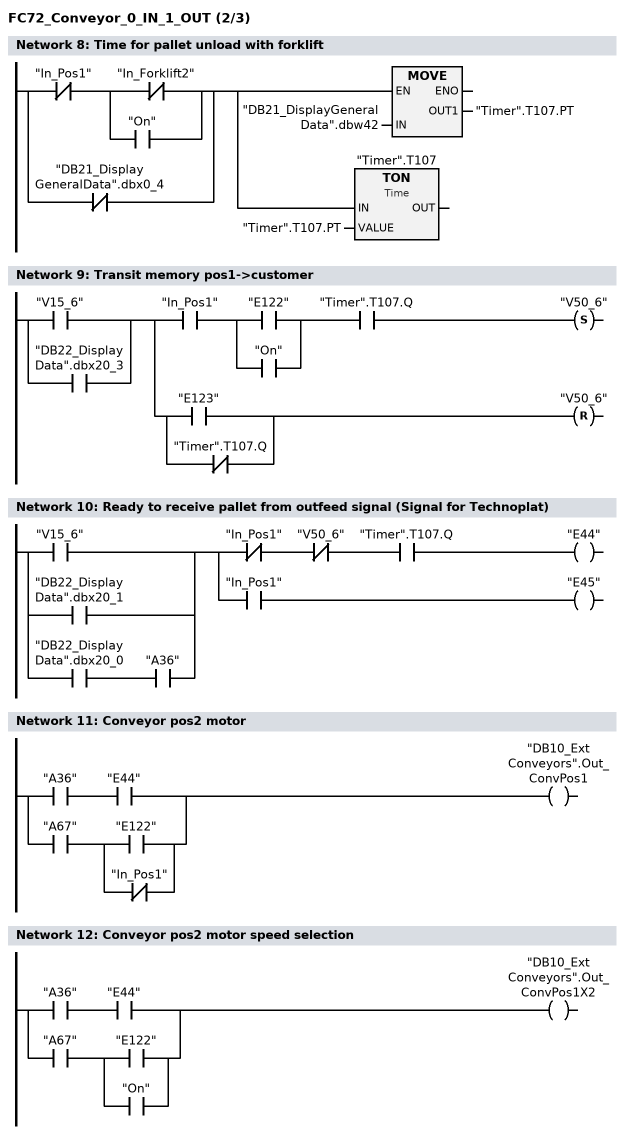
   #_w1 := (NOT "In_Pos1" AND (NOT "In_Forklift2" OR "On")) OR NOT "DB21_DisplayGeneralData".dbx0_4;
   IF #_w1 THEN "Timer".T107.PT := "DB21_DisplayGeneralData".dbw42; END_IF;
   "Timer".T107.TON(IN := #_w1, PT := "Timer".T107.PT);   // TON coil
END_REGION

REGION Network 9: Transit memory pos1->customer
   RUNG wire#powerrail
      Contact( "V15_6" )
      wire#w1
      Contact( "In_Pos1" )
      wire#w2
      Contact( "E122" )
      wire#w3
      Contact( "Timer".T107.Q )
      S_Coil( "V50_6" )
   END_RUNG
   RUNG wire#powerrail
      Contact( "DB22_DisplayData".dbx20_3 )
   END_RUNG wire#w1
   RUNG wire#w2
      Contact( "On" )
   END_RUNG wire#w3
   RUNG wire#w1
      Contact( "E123" )
      wire#w4
      R_Coil( "V50_6" )
   END_RUNG
   RUNG wire#w1
      I_Contact( "Timer".T107.Q )
   END_RUNG wire#w4
   // the same network as SCL:
   #_w1 := "V15_6" OR "DB22_DisplayData".dbx20_3;
   IF #_w1 AND "In_Pos1" AND ("E122" OR "On") AND "Timer".T107.Q THEN "V50_6" := TRUE; END_IF;
   IF #_w1 AND ("E123" OR NOT "Timer".T107.Q) THEN "V50_6" := FALSE; END_IF;
END_REGION

REGION Network 10: Ready to receive pallet from outfeed signal (Signal for Technoplat)
   RUNG wire#powerrail
      Contact( "V15_6" )
      wire#w1
      I_Contact( "In_Pos1" )
      I_Contact( "V50_6" )
      Contact( "Timer".T107.Q )
      Coil( "E44" )
   END_RUNG
   RUNG wire#powerrail
      Contact( "DB22_DisplayData".dbx20_1 )
   END_RUNG wire#w1
   RUNG wire#powerrail
      Contact( "DB22_DisplayData".dbx20_0 )
      Contact( "A36" )
   END_RUNG wire#w1
   RUNG wire#w1
      Contact( "In_Pos1" )
      Coil( "E45" )
   END_RUNG
   // the same network as SCL:
   #_w1 := "V15_6" OR "DB22_DisplayData".dbx20_1 OR ("DB22_DisplayData".dbx20_0 AND "A36");
   "E44" := #_w1 AND NOT "In_Pos1" AND NOT "V50_6" AND "Timer".T107.Q;
   "E45" := #_w1 AND "In_Pos1";
END_REGION

REGION Network 11: Conveyor pos2 motor
   RUNG wire#powerrail
      Contact( "A36" )
      Contact( "E44" )
      wire#w1
      Coil( "DB10_ExtConveyors".Out_ConvPos1 )
   END_RUNG
   RUNG wire#powerrail
      Contact( "A67" )
      wire#w2
      Contact( "E122" )
   END_RUNG wire#w1
   RUNG wire#w2
      I_Contact( "In_Pos1" )
   END_RUNG wire#w1
   // the same network as SCL:
   "DB10_ExtConveyors".Out_ConvPos1 := ("A36" AND "E44") OR ("A67" AND ("E122" OR NOT "In_Pos1"));
END_REGION

REGION Network 12: Conveyor pos2 motor speed selection
   RUNG wire#powerrail
      Contact( "A36" )
      Contact( "E44" )
      wire#w1
      Coil( "DB10_ExtConveyors".Out_ConvPos1X2 )
   END_RUNG
   RUNG wire#powerrail
      Contact( "A67" )
      wire#w2
      Contact( "E122" )
   END_RUNG wire#w1
   RUNG wire#w2
      Contact( "On" )
   END_RUNG wire#w1
   // the same network as SCL:
   "DB10_ExtConveyors".Out_ConvPos1X2 := ("A36" AND "E44") OR ("A67" AND ("E122" OR "On"));
END_REGION

REGION Network 13: Pallet ready in outfeed signal
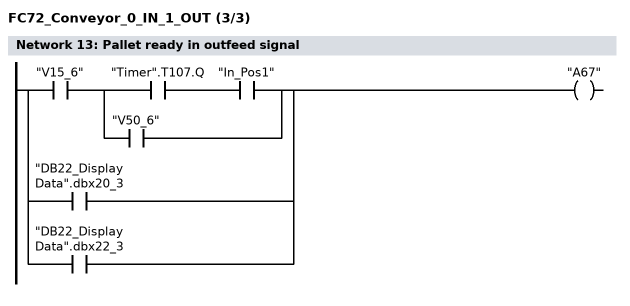
   RUNG wire#powerrail
      Contact( "V15_6" )
      wire#w1
      Contact( "Timer".T107.Q )
      Contact( "In_Pos1" )
      wire#w2
      Coil( "A67" )
   END_RUNG
   RUNG wire#w1
      Contact( "V50_6" )
   END_RUNG wire#w2
   RUNG wire#powerrail
      Contact( "DB22_DisplayData".dbx20_3 )
   END_RUNG wire#w2
   RUNG wire#powerrail
      Contact( "DB22_DisplayData".dbx22_3 )
   END_RUNG wire#w2
   // the same network as SCL:
   "A67" := ("V15_6" AND (("Timer".T107.Q AND "In_Pos1") OR "V50_6")) OR "DB22_DisplayData".dbx20_3 OR "DB22_DisplayData".dbx22_3;
END_REGION
END_FUNCTION

FUNCTION "FC37_MultiprogramSignal" : Void   // FC37, LAD
TITLE = Multiprogram with program selection by external signal
{ S7_Optimized_Access := 'FALSE' }
AUTHOR : Robopac
VERSION : 0.0
// stored: AutoNumber false, IsIECCheckEnabled false, SetENOAutomatically false, UDAEnableTagReadback false
   VAR_TEMP   // added for the SCL form of the ladder/FBD networks
      _w1 : Bool;
   END_VAR
BEGIN

REGION Network 1
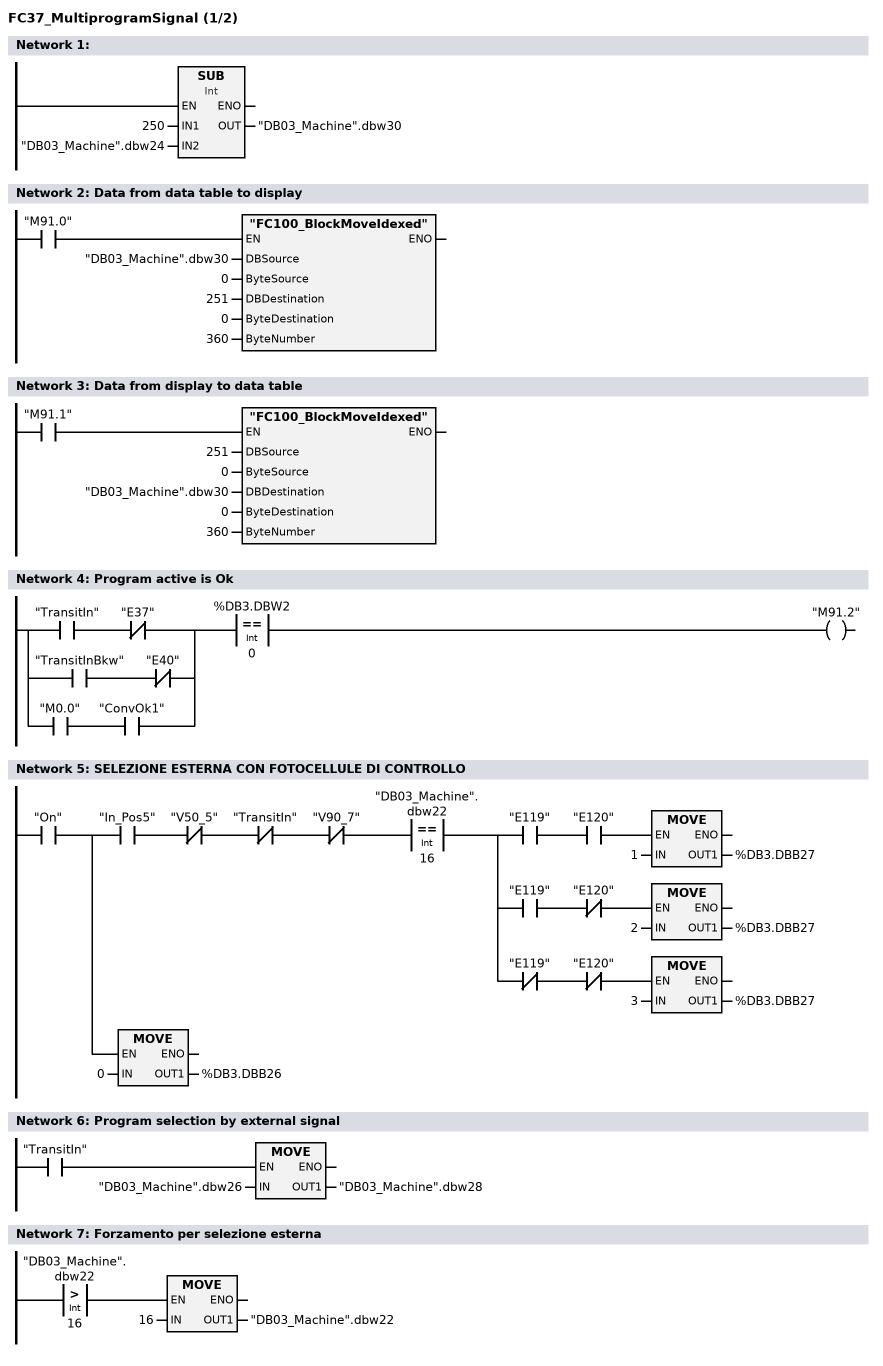
   RUNG wire#powerrail
      { S7_Templates := "SrcType := Int"; S7_GenerateENO := "TRUE" } Sub(in1 := 250, in2 := "DB03_Machine".dbw24, out => "DB03_Machine".dbw30)
   END_RUNG
   // the same network as SCL:
   "DB03_Machine".dbw30 := 250 - "DB03_Machine".dbw24;
END_REGION

REGION Network 2: Data from data table to display
   RUNG wire#powerrail
      Contact( "M91.0" )
      "FC100_BlockMoveIdexed"(DBSource := "DB03_Machine".dbw30, ByteSource := 0, DBDestination := 251, ByteDestination := 0, ByteNumber := 360)
   END_RUNG
   // the same network as SCL:
   IF "M91.0" THEN
       "FC100_BlockMoveIdexed"(DBSource := "DB03_Machine".dbw30,
                               ByteSource := 0,
                               DBDestination := 251,
                               ByteDestination := 0,
                               ByteNumber := 360);
   END_IF;
END_REGION

REGION Network 3: Data from display to data table
   RUNG wire#powerrail
      Contact( "M91.1" )
      "FC100_BlockMoveIdexed"(DBSource := 251, ByteSource := 0, DBDestination := "DB03_Machine".dbw30, ByteDestination := 0, ByteNumber := 360)
   END_RUNG
   // the same network as SCL:
   IF "M91.1" THEN
       "FC100_BlockMoveIdexed"(DBSource := 251,
                               ByteSource := 0,
                               DBDestination := "DB03_Machine".dbw30,
                               ByteDestination := 0,
                               ByteNumber := 360);
   END_IF;
END_REGION

REGION Network 4: Program active is Ok
   RUNG wire#powerrail
      Contact( "TransitIn" )
      I_Contact( "E37" )
      wire#w1
      { S7_Templates := "SrcType := Int" } EQ_Contact(in1 := %DB3.DBW2, in2 := 0)
      Coil( "M91.2" )
   END_RUNG
   RUNG wire#powerrail
      Contact( "TransitInBkw" )
      I_Contact( "E40" )
   END_RUNG wire#w1
   RUNG wire#powerrail
      Contact( "M0.0" )
      Contact( "ConvOk1" )
   END_RUNG wire#w1
   // the same network as SCL:
   "M91.2" := (("TransitIn" AND NOT "E37") OR ("TransitInBkw" AND NOT "E40") OR ("M0.0" AND "ConvOk1")) AND (%DB3.DBW2 = 0);
END_REGION

REGION Network 5: SELEZIONE ESTERNA CON FOTOCELLULE DI CONTROLLO
   RUNG wire#powerrail
      Contact( "On" )
      wire#w1
      Contact( "In_Pos5" )
      I_Contact( "V50_5" )
      I_Contact( "TransitIn" )
      I_Contact( "V90_7" )
      { S7_Templates := "SrcType := Int" } EQ_Contact(in1 := "DB03_Machine".dbw22, in2 := 16)
      wire#w2
      Contact( "E119" )
      Contact( "E120" )
      Move(in := 1, out1 => %DB3.DBB27)
   END_RUNG
   RUNG wire#w2
      Contact( "E119" )
      I_Contact( "E120" )
      Move(in := 2, out1 => %DB3.DBB27)
   END_RUNG
   RUNG wire#w2
      I_Contact( "E119" )
      I_Contact( "E120" )
      Move(in := 3, out1 => %DB3.DBB27)
   END_RUNG
   RUNG wire#w1
      { S7_GenerateENO := "TRUE" } Move(in := 0, out1 => %DB3.DBB26)
   END_RUNG
   // the same network as SCL:
   #_w1 := "On" AND "In_Pos5" AND NOT "V50_5" AND NOT "TransitIn" AND NOT "V90_7" AND ("DB03_Machine".dbw22 = 16);
   IF #_w1 AND "E119" AND "E120" THEN %DB3.DBB27 := 1; END_IF;
   IF #_w1 AND "E119" AND NOT "E120" THEN %DB3.DBB27 := 2; END_IF;
   IF #_w1 AND NOT "E119" AND NOT "E120" THEN %DB3.DBB27 := 3; END_IF;
   IF "On" THEN %DB3.DBB26 := 0; END_IF;
END_REGION

REGION Network 6: Program selection by external signal
   RUNG wire#powerrail
      Contact( "TransitIn" )
      { S7_GenerateENO := "TRUE" } Move(in := "DB03_Machine".dbw26, out1 => "DB03_Machine".dbw28)
   END_RUNG
   // the same network as SCL:
   IF "TransitIn" THEN "DB03_Machine".dbw28 := "DB03_Machine".dbw26; END_IF;
END_REGION

REGION Network 7: Forzamento per selezione esterna
   RUNG wire#powerrail
      { S7_Templates := "SrcType := Int" } GT_Contact(in1 := "DB03_Machine".dbw22, in2 := 16)
      { S7_GenerateENO := "TRUE" } Move(in := 16, out1 => "DB03_Machine".dbw22)
   END_RUNG
   // the same network as SCL:
   IF "DB03_Machine".dbw22 > 16 THEN "DB03_Machine".dbw22 := 16; END_IF;
END_REGION

REGION Network 8: Program selection by display
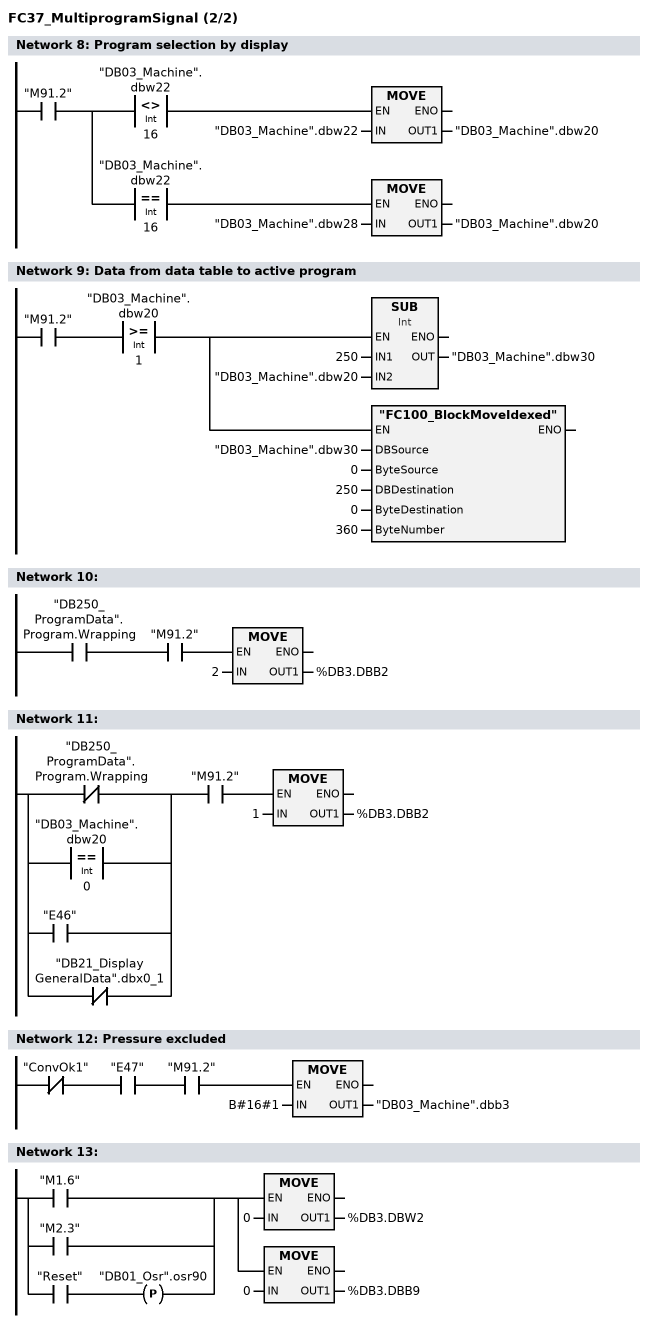
   RUNG wire#powerrail
      Contact( "M91.2" )
      wire#w1
      { S7_Templates := "SrcType := Int" } NE_Contact(in1 := "DB03_Machine".dbw22, in2 := 16)
      { S7_GenerateENO := "TRUE" } Move(in := "DB03_Machine".dbw22, out1 => "DB03_Machine".dbw20)
   END_RUNG
   RUNG wire#w1
      { S7_Templates := "SrcType := Int" } EQ_Contact(in1 := "DB03_Machine".dbw22, in2 := 16)
      { S7_GenerateENO := "TRUE" } Move(in := "DB03_Machine".dbw28, out1 => "DB03_Machine".dbw20)
   END_RUNG
   // the same network as SCL:
   IF "M91.2" AND ("DB03_Machine".dbw22 <> 16) THEN "DB03_Machine".dbw20 := "DB03_Machine".dbw22; END_IF;
   IF "M91.2" AND ("DB03_Machine".dbw22 = 16) THEN "DB03_Machine".dbw20 := "DB03_Machine".dbw28; END_IF;
END_REGION

REGION Network 9: Data from data table to active program
   RUNG wire#powerrail
      Contact( "M91.2" )
      { S7_Templates := "SrcType := Int" } GE_Contact(in1 := "DB03_Machine".dbw20, in2 := 1)
      wire#w1
      { S7_Templates := "SrcType := Int"; S7_GenerateENO := "TRUE" } Sub(in1 := 250, in2 := "DB03_Machine".dbw20, out => "DB03_Machine".dbw30)
   END_RUNG
   RUNG wire#w1
      "FC100_BlockMoveIdexed"(DBSource := "DB03_Machine".dbw30, ByteSource := 0, DBDestination := 250, ByteDestination := 0, ByteNumber := 360)
   END_RUNG
   // the same network as SCL:
   IF "M91.2" AND ("DB03_Machine".dbw20 >= 1) THEN
       "DB03_Machine".dbw30 := 250 - "DB03_Machine".dbw20;
       "FC100_BlockMoveIdexed"(DBSource := "DB03_Machine".dbw30,
                               ByteSource := 0,
                               DBDestination := 250,
                               ByteDestination := 0,
                               ByteNumber := 360);
   END_IF;
END_REGION

REGION Network 10
   RUNG wire#powerrail
      Contact( "DB250_ProgramData".Program.Wrapping )
      Contact( "M91.2" )
      { S7_GenerateENO := "TRUE" } Move(in := 2, out1 => %DB3.DBB2)
   END_RUNG
   // the same network as SCL:
   IF "DB250_ProgramData".Program.Wrapping AND "M91.2" THEN %DB3.DBB2 := 2; END_IF;
END_REGION

REGION Network 11
   RUNG wire#powerrail
      I_Contact( "DB250_ProgramData".Program.Wrapping )
      wire#w1
      Contact( "M91.2" )
      { S7_GenerateENO := "TRUE" } Move(in := 1, out1 => %DB3.DBB2)
   END_RUNG
   RUNG wire#powerrail
      { S7_Templates := "SrcType := Int" } EQ_Contact(in1 := "DB03_Machine".dbw20, in2 := 0)
   END_RUNG wire#w1
   RUNG wire#powerrail
      Contact( "E46" )
   END_RUNG wire#w1
   RUNG wire#powerrail
      I_Contact( "DB21_DisplayGeneralData".dbx0_1 )
   END_RUNG wire#w1
   // the same network as SCL:
   IF (NOT "DB250_ProgramData".Program.Wrapping OR ("DB03_Machine".dbw20 = 0) OR "E46" OR NOT "DB21_DisplayGeneralData".dbx0_1) AND "M91.2" THEN
       %DB3.DBB2 := 1;
   END_IF;
END_REGION

REGION Network 12: Pressure excluded
   RUNG wire#powerrail
      I_Contact( "ConvOk1" )
      Contact( "E47" )
      Contact( "M91.2" )
      { S7_GenerateENO := "TRUE" } Move(in := B#16#1, out1 => "DB03_Machine".dbb3)
   END_RUNG
   // the same network as SCL:
   IF NOT "ConvOk1" AND "E47" AND "M91.2" THEN "DB03_Machine".dbb3 := B#16#1; END_IF;
END_REGION

REGION Network 13
   RUNG wire#powerrail
      Contact( "M1.6" )
      wire#w1
      { S7_GenerateENO := "TRUE" } Move(in := 0, out1 => %DB3.DBW2)
   END_RUNG
   RUNG wire#powerrail
      Contact( "M2.3" )
   END_RUNG wire#w1
   RUNG wire#powerrail
      Contact( "Reset" )
      P_Trig( "DB01_Osr".osr90 )
   END_RUNG wire#w1
   RUNG wire#w1
      { S7_GenerateENO := "TRUE" } Move(in := 0, out1 => %DB3.DBB9)
   END_RUNG
   // the same network as SCL:
   #_w1 := "Reset" AND NOT "DB01_Osr".osr90;   // rising edge
   "DB01_Osr".osr90 := "Reset";
   IF "M1.6" OR "M2.3" OR #_w1 THEN
       %DB3.DBW2 := 0;
       %DB3.DBB9 := 0;
   END_IF;
END_REGION
END_FUNCTION

FUNCTION "FC39_DisplaySiemensTP" : Void   // FC39, LAD
TITLE = Display Siemens TP177 management
{ S7_Optimized_Access := 'FALSE' }
AUTHOR : Robopac
VERSION : 0.0
// stored: AutoNumber false, IsIECCheckEnabled false, SetENOAutomatically false, UDAEnableTagReadback false
   VAR_TEMP
      TempInt : Int;
   END_VAR
   VAR_TEMP   // added for the SCL form of the ladder/FBD networks
      _w1 : Bool;
      _w2 : Bool;
      _w3 : Bool;
      _w4 : Bool;
      _w5 : Bool;
      _w6 : Bool;
   END_VAR
BEGIN

REGION Network 1: Manual(Toggle bit): Pressure plate upward/downward (Helix)
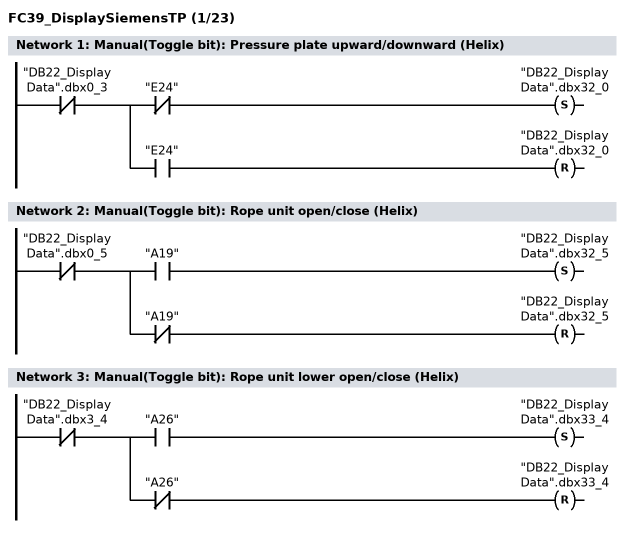
   RUNG wire#powerrail
      I_Contact( "DB22_DisplayData".dbx0_3 )
      wire#w1
      I_Contact( "E24" )
      S_Coil( "DB22_DisplayData".dbx32_0 )
   END_RUNG
   RUNG wire#w1
      Contact( "E24" )
      R_Coil( "DB22_DisplayData".dbx32_0 )
   END_RUNG
   // the same network as SCL:
   #_w1 := NOT "DB22_DisplayData".dbx0_3;
   IF #_w1 AND NOT "E24" THEN "DB22_DisplayData".dbx32_0 := TRUE; END_IF;
   IF #_w1 AND "E24" THEN "DB22_DisplayData".dbx32_0 := FALSE; END_IF;
END_REGION

REGION Network 2: Manual(Toggle bit): Rope unit open/close (Helix)
   RUNG wire#powerrail
      I_Contact( "DB22_DisplayData".dbx0_5 )
      wire#w1
      Contact( "A19" )
      S_Coil( "DB22_DisplayData".dbx32_5 )
   END_RUNG
   RUNG wire#w1
      I_Contact( "A19" )
      R_Coil( "DB22_DisplayData".dbx32_5 )
   END_RUNG
   // the same network as SCL:
   #_w1 := NOT "DB22_DisplayData".dbx0_5;
   IF #_w1 AND "A19" THEN "DB22_DisplayData".dbx32_5 := TRUE; END_IF;
   IF #_w1 AND NOT "A19" THEN "DB22_DisplayData".dbx32_5 := FALSE; END_IF;
END_REGION

REGION Network 3: Manual(Toggle bit): Rope unit lower open/close (Helix)
   RUNG wire#powerrail
      I_Contact( "DB22_DisplayData".dbx3_4 )
      wire#w1
      Contact( "A26" )
      S_Coil( "DB22_DisplayData".dbx33_4 )
   END_RUNG
   RUNG wire#w1
      I_Contact( "A26" )
      R_Coil( "DB22_DisplayData".dbx33_4 )
   END_RUNG
   // the same network as SCL:
   #_w1 := NOT "DB22_DisplayData".dbx3_4;
   IF #_w1 AND "A26" THEN "DB22_DisplayData".dbx33_4 := TRUE; END_IF;
   IF #_w1 AND NOT "A26" THEN "DB22_DisplayData".dbx33_4 := FALSE; END_IF;
END_REGION

REGION Network 4: Manual operation for Helix
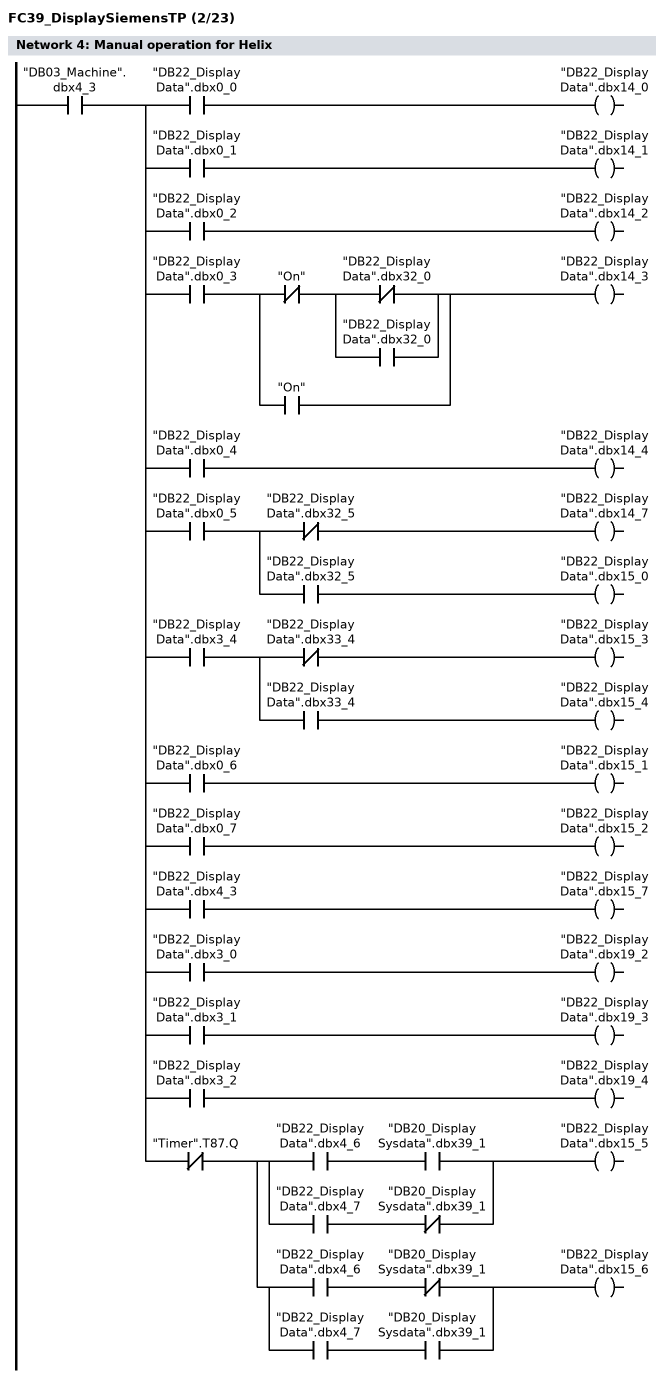
   RUNG wire#powerrail
      Contact( "DB03_Machine".dbx4_3 )
      wire#w1
      Contact( "DB22_DisplayData".dbx0_0 )
      Coil( "DB22_DisplayData".dbx14_0 )
   END_RUNG
   RUNG wire#w1
      Contact( "DB22_DisplayData".dbx0_1 )
      Coil( "DB22_DisplayData".dbx14_1 )
   END_RUNG
   RUNG wire#w1
      Contact( "DB22_DisplayData".dbx0_2 )
      Coil( "DB22_DisplayData".dbx14_2 )
   END_RUNG
   RUNG wire#w1
      Contact( "DB22_DisplayData".dbx0_3 )
      wire#w2
      I_Contact( "On" )
      wire#w3
      I_Contact( "DB22_DisplayData".dbx32_0 )
      wire#w4
      Coil( "DB22_DisplayData".dbx14_3 )
   END_RUNG
   RUNG wire#w3
      Contact( "DB22_DisplayData".dbx32_0 )
   END_RUNG wire#w4
   RUNG wire#w2
      Contact( "On" )
   END_RUNG wire#w4
   RUNG wire#w1
      Contact( "DB22_DisplayData".dbx0_4 )
      Coil( "DB22_DisplayData".dbx14_4 )
   END_RUNG
   RUNG wire#w1
      Contact( "DB22_DisplayData".dbx0_5 )
      wire#w5
      I_Contact( "DB22_DisplayData".dbx32_5 )
      Coil( "DB22_DisplayData".dbx14_7 )
   END_RUNG
   RUNG wire#w5
      Contact( "DB22_DisplayData".dbx32_5 )
      Coil( "DB22_DisplayData".dbx15_0 )
   END_RUNG
   RUNG wire#w1
      Contact( "DB22_DisplayData".dbx3_4 )
      wire#w6
      I_Contact( "DB22_DisplayData".dbx33_4 )
      Coil( "DB22_DisplayData".dbx15_3 )
   END_RUNG
   RUNG wire#w6
      Contact( "DB22_DisplayData".dbx33_4 )
      Coil( "DB22_DisplayData".dbx15_4 )
   END_RUNG
   RUNG wire#w1
      Contact( "DB22_DisplayData".dbx0_6 )
      Coil( "DB22_DisplayData".dbx15_1 )
   END_RUNG
   RUNG wire#w1
      Contact( "DB22_DisplayData".dbx0_7 )
      Coil( "DB22_DisplayData".dbx15_2 )
   END_RUNG
   RUNG wire#w1
      Contact( "DB22_DisplayData".dbx4_3 )
      Coil( "DB22_DisplayData".dbx15_7 )
   END_RUNG
   RUNG wire#w1
      Contact( "DB22_DisplayData".dbx3_0 )
      Coil( "DB22_DisplayData".dbx19_2 )
   END_RUNG
   RUNG wire#w1
      Contact( "DB22_DisplayData".dbx3_1 )
      Coil( "DB22_DisplayData".dbx19_3 )
   END_RUNG
   RUNG wire#w1
      Contact( "DB22_DisplayData".dbx3_2 )
      Coil( "DB22_DisplayData".dbx19_4 )
   END_RUNG
   RUNG wire#w1
      I_Contact( "Timer".T87.Q )
      wire#w7
      Contact( "DB22_DisplayData".dbx4_6 )
      Contact( "DB20_DisplaySysdata".dbx39_1 )
      wire#w8
      Coil( "DB22_DisplayData".dbx15_5 )
   END_RUNG
   RUNG wire#w7
      Contact( "DB22_DisplayData".dbx4_7 )
      I_Contact( "DB20_DisplaySysdata".dbx39_1 )
   END_RUNG wire#w8
   RUNG wire#w7
      Contact( "DB22_DisplayData".dbx4_6 )
      I_Contact( "DB20_DisplaySysdata".dbx39_1 )
      wire#w9
      Coil( "DB22_DisplayData".dbx15_6 )
   END_RUNG
   RUNG wire#w7
      Contact( "DB22_DisplayData".dbx4_7 )
      Contact( "DB20_DisplaySysdata".dbx39_1 )
   END_RUNG wire#w9
   // the same network as SCL:
   "DB22_DisplayData".dbx14_0 := "DB03_Machine".dbx4_3 AND "DB22_DisplayData".dbx0_0;
   "DB22_DisplayData".dbx14_1 := "DB03_Machine".dbx4_3 AND "DB22_DisplayData".dbx0_1;
   "DB22_DisplayData".dbx14_2 := "DB03_Machine".dbx4_3 AND "DB22_DisplayData".dbx0_2;
   "DB22_DisplayData".dbx14_3 := "DB03_Machine".dbx4_3 AND "DB22_DisplayData".dbx0_3 AND ((NOT "On" AND (NOT "DB22_DisplayData".dbx32_0 OR "DB22_DisplayData".dbx32_0)) OR "On");
   "DB22_DisplayData".dbx14_4 := "DB03_Machine".dbx4_3 AND "DB22_DisplayData".dbx0_4;
   #_w1 := "DB03_Machine".dbx4_3 AND "DB22_DisplayData".dbx0_5;
   "DB22_DisplayData".dbx14_7 := #_w1 AND NOT "DB22_DisplayData".dbx32_5;
   "DB22_DisplayData".dbx15_0 := #_w1 AND "DB22_DisplayData".dbx32_5;
   #_w2 := "DB03_Machine".dbx4_3 AND "DB22_DisplayData".dbx3_4;
   "DB22_DisplayData".dbx15_3 := #_w2 AND NOT "DB22_DisplayData".dbx33_4;
   "DB22_DisplayData".dbx15_4 := #_w2 AND "DB22_DisplayData".dbx33_4;
   "DB22_DisplayData".dbx15_1 := "DB03_Machine".dbx4_3 AND "DB22_DisplayData".dbx0_6;
   "DB22_DisplayData".dbx15_2 := "DB03_Machine".dbx4_3 AND "DB22_DisplayData".dbx0_7;
   "DB22_DisplayData".dbx15_7 := "DB03_Machine".dbx4_3 AND "DB22_DisplayData".dbx4_3;
   "DB22_DisplayData".dbx19_2 := "DB03_Machine".dbx4_3 AND "DB22_DisplayData".dbx3_0;
   "DB22_DisplayData".dbx19_3 := "DB03_Machine".dbx4_3 AND "DB22_DisplayData".dbx3_1;
   "DB22_DisplayData".dbx19_4 := "DB03_Machine".dbx4_3 AND "DB22_DisplayData".dbx3_2;
   #_w3 := "DB03_Machine".dbx4_3 AND NOT "Timer".T87.Q;
   "DB22_DisplayData".dbx15_5 := #_w3 AND (("DB22_DisplayData".dbx4_6 AND "DB20_DisplaySysdata".dbx39_1) OR ("DB22_DisplayData".dbx4_7 AND NOT "DB20_DisplaySysdata".dbx39_1));
   "DB22_DisplayData".dbx15_6 := #_w3 AND (("DB22_DisplayData".dbx4_6 AND NOT "DB20_DisplaySysdata".dbx39_1) OR ("DB22_DisplayData".dbx4_7 AND "DB20_DisplaySysdata".dbx39_1));
END_REGION

REGION Network 5: Manual(Toggle bit): Clamp upward/downward (Clamp)
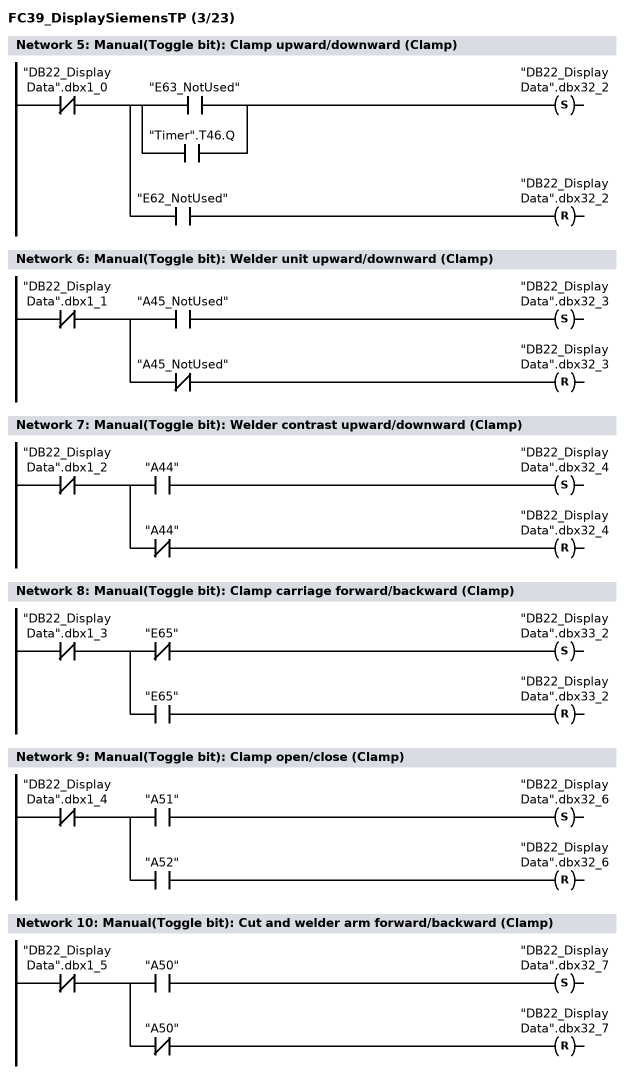
   RUNG wire#powerrail
      I_Contact( "DB22_DisplayData".dbx1_0 )
      wire#w1
      Contact( "E63_NotUsed" )
      wire#w2
      S_Coil( "DB22_DisplayData".dbx32_2 )
   END_RUNG
   RUNG wire#w1
      Contact( "Timer".T46.Q )
   END_RUNG wire#w2
   RUNG wire#w1
      Contact( "E62_NotUsed" )
      R_Coil( "DB22_DisplayData".dbx32_2 )
   END_RUNG
   // the same network as SCL:
   #_w1 := NOT "DB22_DisplayData".dbx1_0;
   IF #_w1 AND ("E63_NotUsed" OR "Timer".T46.Q) THEN "DB22_DisplayData".dbx32_2 := TRUE; END_IF;
   IF #_w1 AND "E62_NotUsed" THEN "DB22_DisplayData".dbx32_2 := FALSE; END_IF;
END_REGION

REGION Network 6: Manual(Toggle bit): Welder unit upward/downward (Clamp)
   RUNG wire#powerrail
      I_Contact( "DB22_DisplayData".dbx1_1 )
      wire#w1
      Contact( "A45_NotUsed" )
      S_Coil( "DB22_DisplayData".dbx32_3 )
   END_RUNG
   RUNG wire#w1
      I_Contact( "A45_NotUsed" )
      R_Coil( "DB22_DisplayData".dbx32_3 )
   END_RUNG
   // the same network as SCL:
   #_w1 := NOT "DB22_DisplayData".dbx1_1;
   IF #_w1 AND "A45_NotUsed" THEN "DB22_DisplayData".dbx32_3 := TRUE; END_IF;
   IF #_w1 AND NOT "A45_NotUsed" THEN "DB22_DisplayData".dbx32_3 := FALSE; END_IF;
END_REGION

REGION Network 7: Manual(Toggle bit): Welder contrast upward/downward (Clamp)
   RUNG wire#powerrail
      I_Contact( "DB22_DisplayData".dbx1_2 )
      wire#w1
      Contact( "A44" )
      S_Coil( "DB22_DisplayData".dbx32_4 )
   END_RUNG
   RUNG wire#w1
      I_Contact( "A44" )
      R_Coil( "DB22_DisplayData".dbx32_4 )
   END_RUNG
   // the same network as SCL:
   #_w1 := NOT "DB22_DisplayData".dbx1_2;
   IF #_w1 AND "A44" THEN "DB22_DisplayData".dbx32_4 := TRUE; END_IF;
   IF #_w1 AND NOT "A44" THEN "DB22_DisplayData".dbx32_4 := FALSE; END_IF;
END_REGION

REGION Network 8: Manual(Toggle bit): Clamp carriage forward/backward (Clamp)
   RUNG wire#powerrail
      I_Contact( "DB22_DisplayData".dbx1_3 )
      wire#w1
      I_Contact( "E65" )
      S_Coil( "DB22_DisplayData".dbx33_2 )
   END_RUNG
   RUNG wire#w1
      Contact( "E65" )
      R_Coil( "DB22_DisplayData".dbx33_2 )
   END_RUNG
   // the same network as SCL:
   #_w1 := NOT "DB22_DisplayData".dbx1_3;
   IF #_w1 AND NOT "E65" THEN "DB22_DisplayData".dbx33_2 := TRUE; END_IF;
   IF #_w1 AND "E65" THEN "DB22_DisplayData".dbx33_2 := FALSE; END_IF;
END_REGION

REGION Network 9: Manual(Toggle bit): Clamp open/close (Clamp)
   RUNG wire#powerrail
      I_Contact( "DB22_DisplayData".dbx1_4 )
      wire#w1
      Contact( "A51" )
      S_Coil( "DB22_DisplayData".dbx32_6 )
   END_RUNG
   RUNG wire#w1
      Contact( "A52" )
      R_Coil( "DB22_DisplayData".dbx32_6 )
   END_RUNG
   // the same network as SCL:
   #_w1 := NOT "DB22_DisplayData".dbx1_4;
   IF #_w1 AND "A51" THEN "DB22_DisplayData".dbx32_6 := TRUE; END_IF;
   IF #_w1 AND "A52" THEN "DB22_DisplayData".dbx32_6 := FALSE; END_IF;
END_REGION

REGION Network 10: Manual(Toggle bit): Cut and welder arm forward/backward (Clamp)
   RUNG wire#powerrail
      I_Contact( "DB22_DisplayData".dbx1_5 )
      wire#w1
      Contact( "A50" )
      S_Coil( "DB22_DisplayData".dbx32_7 )
   END_RUNG
   RUNG wire#w1
      I_Contact( "A50" )
      R_Coil( "DB22_DisplayData".dbx32_7 )
   END_RUNG
   // the same network as SCL:
   #_w1 := NOT "DB22_DisplayData".dbx1_5;
   IF #_w1 AND "A50" THEN "DB22_DisplayData".dbx32_7 := TRUE; END_IF;
   IF #_w1 AND NOT "A50" THEN "DB22_DisplayData".dbx32_7 := FALSE; END_IF;
END_REGION

REGION Network 11: Manual operation for clamp unit
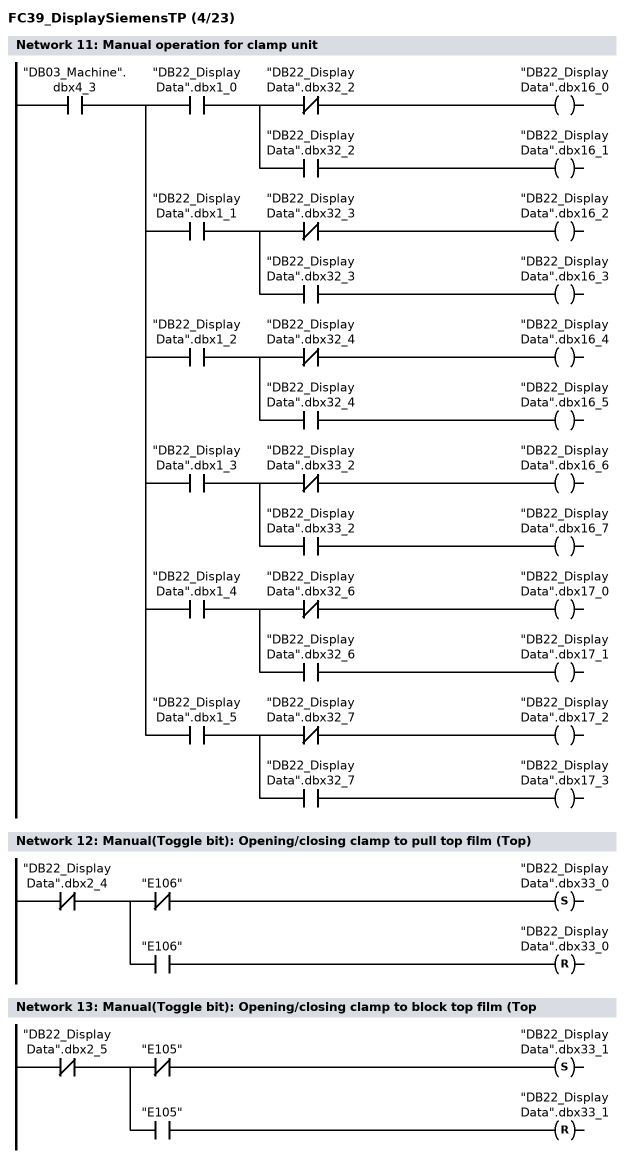
   RUNG wire#powerrail
      Contact( "DB03_Machine".dbx4_3 )
      wire#w1
      Contact( "DB22_DisplayData".dbx1_0 )
      wire#w2
      I_Contact( "DB22_DisplayData".dbx32_2 )
      Coil( "DB22_DisplayData".dbx16_0 )
   END_RUNG
   RUNG wire#w2
      Contact( "DB22_DisplayData".dbx32_2 )
      Coil( "DB22_DisplayData".dbx16_1 )
   END_RUNG
   RUNG wire#w1
      Contact( "DB22_DisplayData".dbx1_1 )
      wire#w3
      I_Contact( "DB22_DisplayData".dbx32_3 )
      Coil( "DB22_DisplayData".dbx16_2 )
   END_RUNG
   RUNG wire#w3
      Contact( "DB22_DisplayData".dbx32_3 )
      Coil( "DB22_DisplayData".dbx16_3 )
   END_RUNG
   RUNG wire#w1
      Contact( "DB22_DisplayData".dbx1_2 )
      wire#w4
      I_Contact( "DB22_DisplayData".dbx32_4 )
      Coil( "DB22_DisplayData".dbx16_4 )
   END_RUNG
   RUNG wire#w4
      Contact( "DB22_DisplayData".dbx32_4 )
      Coil( "DB22_DisplayData".dbx16_5 )
   END_RUNG
   RUNG wire#w1
      Contact( "DB22_DisplayData".dbx1_3 )
      wire#w5
      I_Contact( "DB22_DisplayData".dbx33_2 )
      Coil( "DB22_DisplayData".dbx16_6 )
   END_RUNG
   RUNG wire#w5
      Contact( "DB22_DisplayData".dbx33_2 )
      Coil( "DB22_DisplayData".dbx16_7 )
   END_RUNG
   RUNG wire#w1
      Contact( "DB22_DisplayData".dbx1_4 )
      wire#w6
      I_Contact( "DB22_DisplayData".dbx32_6 )
      Coil( "DB22_DisplayData".dbx17_0 )
   END_RUNG
   RUNG wire#w6
      Contact( "DB22_DisplayData".dbx32_6 )
      Coil( "DB22_DisplayData".dbx17_1 )
   END_RUNG
   RUNG wire#w1
      Contact( "DB22_DisplayData".dbx1_5 )
      wire#w7
      I_Contact( "DB22_DisplayData".dbx32_7 )
      Coil( "DB22_DisplayData".dbx17_2 )
   END_RUNG
   RUNG wire#w7
      Contact( "DB22_DisplayData".dbx32_7 )
      Coil( "DB22_DisplayData".dbx17_3 )
   END_RUNG
   // the same network as SCL:
   #_w1 := "DB03_Machine".dbx4_3 AND "DB22_DisplayData".dbx1_0;
   "DB22_DisplayData".dbx16_0 := #_w1 AND NOT "DB22_DisplayData".dbx32_2;
   "DB22_DisplayData".dbx16_1 := #_w1 AND "DB22_DisplayData".dbx32_2;
   #_w2 := "DB03_Machine".dbx4_3 AND "DB22_DisplayData".dbx1_1;
   "DB22_DisplayData".dbx16_2 := #_w2 AND NOT "DB22_DisplayData".dbx32_3;
   "DB22_DisplayData".dbx16_3 := #_w2 AND "DB22_DisplayData".dbx32_3;
   #_w3 := "DB03_Machine".dbx4_3 AND "DB22_DisplayData".dbx1_2;
   "DB22_DisplayData".dbx16_4 := #_w3 AND NOT "DB22_DisplayData".dbx32_4;
   "DB22_DisplayData".dbx16_5 := #_w3 AND "DB22_DisplayData".dbx32_4;
   #_w4 := "DB03_Machine".dbx4_3 AND "DB22_DisplayData".dbx1_3;
   "DB22_DisplayData".dbx16_6 := #_w4 AND NOT "DB22_DisplayData".dbx33_2;
   "DB22_DisplayData".dbx16_7 := #_w4 AND "DB22_DisplayData".dbx33_2;
   #_w5 := "DB03_Machine".dbx4_3 AND "DB22_DisplayData".dbx1_4;
   "DB22_DisplayData".dbx17_0 := #_w5 AND NOT "DB22_DisplayData".dbx32_6;
   "DB22_DisplayData".dbx17_1 := #_w5 AND "DB22_DisplayData".dbx32_6;
   #_w6 := "DB03_Machine".dbx4_3 AND "DB22_DisplayData".dbx1_5;
   "DB22_DisplayData".dbx17_2 := #_w6 AND NOT "DB22_DisplayData".dbx32_7;
   "DB22_DisplayData".dbx17_3 := #_w6 AND "DB22_DisplayData".dbx32_7;
END_REGION

REGION Network 12: Manual(Toggle bit): Opening/closing clamp to pull top film (Top)
   RUNG wire#powerrail
      I_Contact( "DB22_DisplayData".dbx2_4 )
      wire#w1
      I_Contact( "E106" )
      S_Coil( "DB22_DisplayData".dbx33_0 )
   END_RUNG
   RUNG wire#w1
      Contact( "E106" )
      R_Coil( "DB22_DisplayData".dbx33_0 )
   END_RUNG
   // the same network as SCL:
   #_w1 := NOT "DB22_DisplayData".dbx2_4;
   IF #_w1 AND NOT "E106" THEN "DB22_DisplayData".dbx33_0 := TRUE; END_IF;
   IF #_w1 AND "E106" THEN "DB22_DisplayData".dbx33_0 := FALSE; END_IF;
END_REGION

REGION Network 13: Manual(Toggle bit): Opening/closing clamp to block top film (Top
   RUNG wire#powerrail
      I_Contact( "DB22_DisplayData".dbx2_5 )
      wire#w1
      I_Contact( "E105" )
      S_Coil( "DB22_DisplayData".dbx33_1 )
   END_RUNG
   RUNG wire#w1
      Contact( "E105" )
      R_Coil( "DB22_DisplayData".dbx33_1 )
   END_RUNG
   // the same network as SCL:
   #_w1 := NOT "DB22_DisplayData".dbx2_5;
   IF #_w1 AND NOT "E105" THEN "DB22_DisplayData".dbx33_1 := TRUE; END_IF;
   IF #_w1 AND "E105" THEN "DB22_DisplayData".dbx33_1 := FALSE; END_IF;
END_REGION

REGION Network 14: Maual operation for top unit
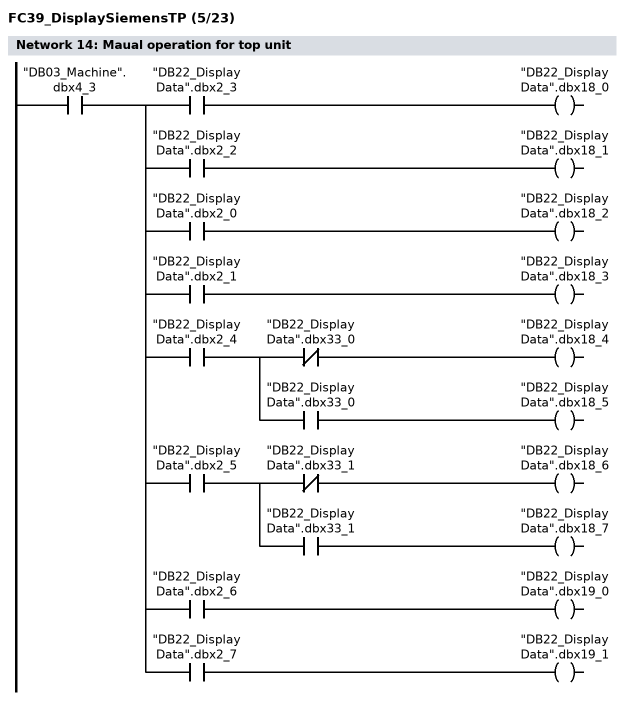
   RUNG wire#powerrail
      Contact( "DB03_Machine".dbx4_3 )
      wire#w1
      Contact( "DB22_DisplayData".dbx2_3 )
      Coil( "DB22_DisplayData".dbx18_0 )
   END_RUNG
   RUNG wire#w1
      Contact( "DB22_DisplayData".dbx2_2 )
      Coil( "DB22_DisplayData".dbx18_1 )
   END_RUNG
   RUNG wire#w1
      Contact( "DB22_DisplayData".dbx2_0 )
      Coil( "DB22_DisplayData".dbx18_2 )
   END_RUNG
   RUNG wire#w1
      Contact( "DB22_DisplayData".dbx2_1 )
      Coil( "DB22_DisplayData".dbx18_3 )
   END_RUNG
   RUNG wire#w1
      Contact( "DB22_DisplayData".dbx2_4 )
      wire#w2
      I_Contact( "DB22_DisplayData".dbx33_0 )
      Coil( "DB22_DisplayData".dbx18_4 )
   END_RUNG
   RUNG wire#w2
      Contact( "DB22_DisplayData".dbx33_0 )
      Coil( "DB22_DisplayData".dbx18_5 )
   END_RUNG
   RUNG wire#w1
      Contact( "DB22_DisplayData".dbx2_5 )
      wire#w3
      I_Contact( "DB22_DisplayData".dbx33_1 )
      Coil( "DB22_DisplayData".dbx18_6 )
   END_RUNG
   RUNG wire#w3
      Contact( "DB22_DisplayData".dbx33_1 )
      Coil( "DB22_DisplayData".dbx18_7 )
   END_RUNG
   RUNG wire#w1
      Contact( "DB22_DisplayData".dbx2_6 )
      Coil( "DB22_DisplayData".dbx19_0 )
   END_RUNG
   RUNG wire#w1
      Contact( "DB22_DisplayData".dbx2_7 )
      Coil( "DB22_DisplayData".dbx19_1 )
   END_RUNG
   // the same network as SCL:
   "DB22_DisplayData".dbx18_0 := "DB03_Machine".dbx4_3 AND "DB22_DisplayData".dbx2_3;
   "DB22_DisplayData".dbx18_1 := "DB03_Machine".dbx4_3 AND "DB22_DisplayData".dbx2_2;
   "DB22_DisplayData".dbx18_2 := "DB03_Machine".dbx4_3 AND "DB22_DisplayData".dbx2_0;
   "DB22_DisplayData".dbx18_3 := "DB03_Machine".dbx4_3 AND "DB22_DisplayData".dbx2_1;
   #_w1 := "DB03_Machine".dbx4_3 AND "DB22_DisplayData".dbx2_4;
   "DB22_DisplayData".dbx18_4 := #_w1 AND NOT "DB22_DisplayData".dbx33_0;
   "DB22_DisplayData".dbx18_5 := #_w1 AND "DB22_DisplayData".dbx33_0;
   #_w2 := "DB03_Machine".dbx4_3 AND "DB22_DisplayData".dbx2_5;
   "DB22_DisplayData".dbx18_6 := #_w2 AND NOT "DB22_DisplayData".dbx33_1;
   "DB22_DisplayData".dbx18_7 := #_w2 AND "DB22_DisplayData".dbx33_1;
   "DB22_DisplayData".dbx19_0 := "DB03_Machine".dbx4_3 AND "DB22_DisplayData".dbx2_6;
   "DB22_DisplayData".dbx19_1 := "DB03_Machine".dbx4_3 AND "DB22_DisplayData".dbx2_7;
END_REGION

REGION Network 15: Diagnostic signal conveyor
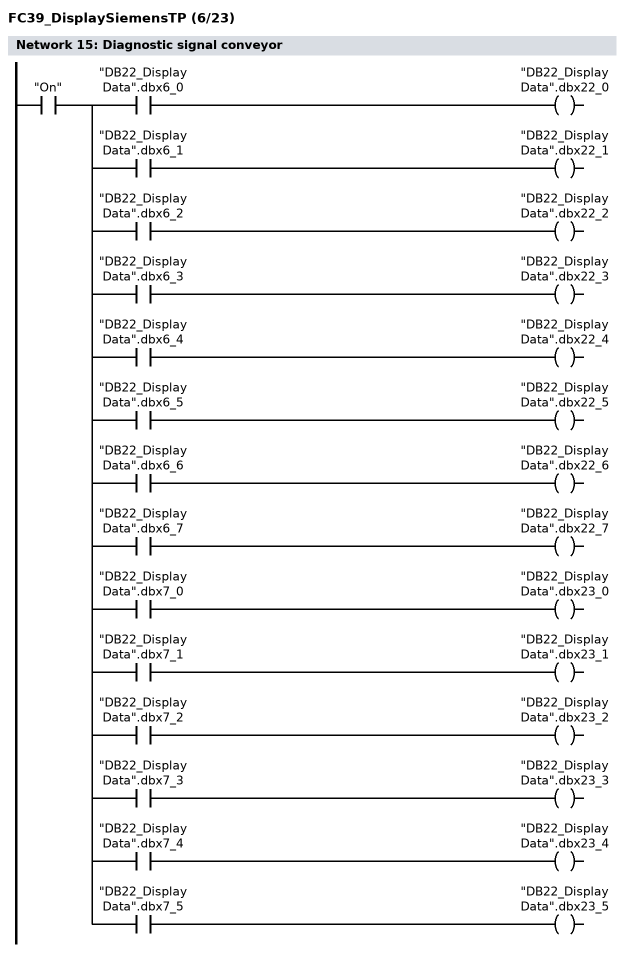
   RUNG wire#powerrail
      Contact( "On" )
      wire#w1
      Contact( "DB22_DisplayData".dbx6_0 )
      Coil( "DB22_DisplayData".dbx22_0 )
   END_RUNG
   RUNG wire#w1
      Contact( "DB22_DisplayData".dbx6_1 )
      Coil( "DB22_DisplayData".dbx22_1 )
   END_RUNG
   RUNG wire#w1
      Contact( "DB22_DisplayData".dbx6_2 )
      Coil( "DB22_DisplayData".dbx22_2 )
   END_RUNG
   RUNG wire#w1
      Contact( "DB22_DisplayData".dbx6_3 )
      Coil( "DB22_DisplayData".dbx22_3 )
   END_RUNG
   RUNG wire#w1
      Contact( "DB22_DisplayData".dbx6_4 )
      Coil( "DB22_DisplayData".dbx22_4 )
   END_RUNG
   RUNG wire#w1
      Contact( "DB22_DisplayData".dbx6_5 )
      Coil( "DB22_DisplayData".dbx22_5 )
   END_RUNG
   RUNG wire#w1
      Contact( "DB22_DisplayData".dbx6_6 )
      Coil( "DB22_DisplayData".dbx22_6 )
   END_RUNG
   RUNG wire#w1
      Contact( "DB22_DisplayData".dbx6_7 )
      Coil( "DB22_DisplayData".dbx22_7 )
   END_RUNG
   RUNG wire#w1
      Contact( "DB22_DisplayData".dbx7_0 )
      Coil( "DB22_DisplayData".dbx23_0 )
   END_RUNG
   RUNG wire#w1
      Contact( "DB22_DisplayData".dbx7_1 )
      Coil( "DB22_DisplayData".dbx23_1 )
   END_RUNG
   RUNG wire#w1
      Contact( "DB22_DisplayData".dbx7_2 )
      Coil( "DB22_DisplayData".dbx23_2 )
   END_RUNG
   RUNG wire#w1
      Contact( "DB22_DisplayData".dbx7_3 )
      Coil( "DB22_DisplayData".dbx23_3 )
   END_RUNG
   RUNG wire#w1
      Contact( "DB22_DisplayData".dbx7_4 )
      Coil( "DB22_DisplayData".dbx23_4 )
   END_RUNG
   RUNG wire#w1
      Contact( "DB22_DisplayData".dbx7_5 )
      Coil( "DB22_DisplayData".dbx23_5 )
   END_RUNG
   // the same network as SCL:
   "DB22_DisplayData".dbx22_0 := "On" AND "DB22_DisplayData".dbx6_0;
   "DB22_DisplayData".dbx22_1 := "On" AND "DB22_DisplayData".dbx6_1;
   "DB22_DisplayData".dbx22_2 := "On" AND "DB22_DisplayData".dbx6_2;
   "DB22_DisplayData".dbx22_3 := "On" AND "DB22_DisplayData".dbx6_3;
   "DB22_DisplayData".dbx22_4 := "On" AND "DB22_DisplayData".dbx6_4;
   "DB22_DisplayData".dbx22_5 := "On" AND "DB22_DisplayData".dbx6_5;
   "DB22_DisplayData".dbx22_6 := "On" AND "DB22_DisplayData".dbx6_6;
   "DB22_DisplayData".dbx22_7 := "On" AND "DB22_DisplayData".dbx6_7;
   "DB22_DisplayData".dbx23_0 := "On" AND "DB22_DisplayData".dbx7_0;
   "DB22_DisplayData".dbx23_1 := "On" AND "DB22_DisplayData".dbx7_1;
   "DB22_DisplayData".dbx23_2 := "On" AND "DB22_DisplayData".dbx7_2;
   "DB22_DisplayData".dbx23_3 := "On" AND "DB22_DisplayData".dbx7_3;
   "DB22_DisplayData".dbx23_4 := "On" AND "DB22_DisplayData".dbx7_4;
   "DB22_DisplayData".dbx23_5 := "On" AND "DB22_DisplayData".dbx7_5;
END_REGION

REGION Network 16: Diagnostic signal conveyor
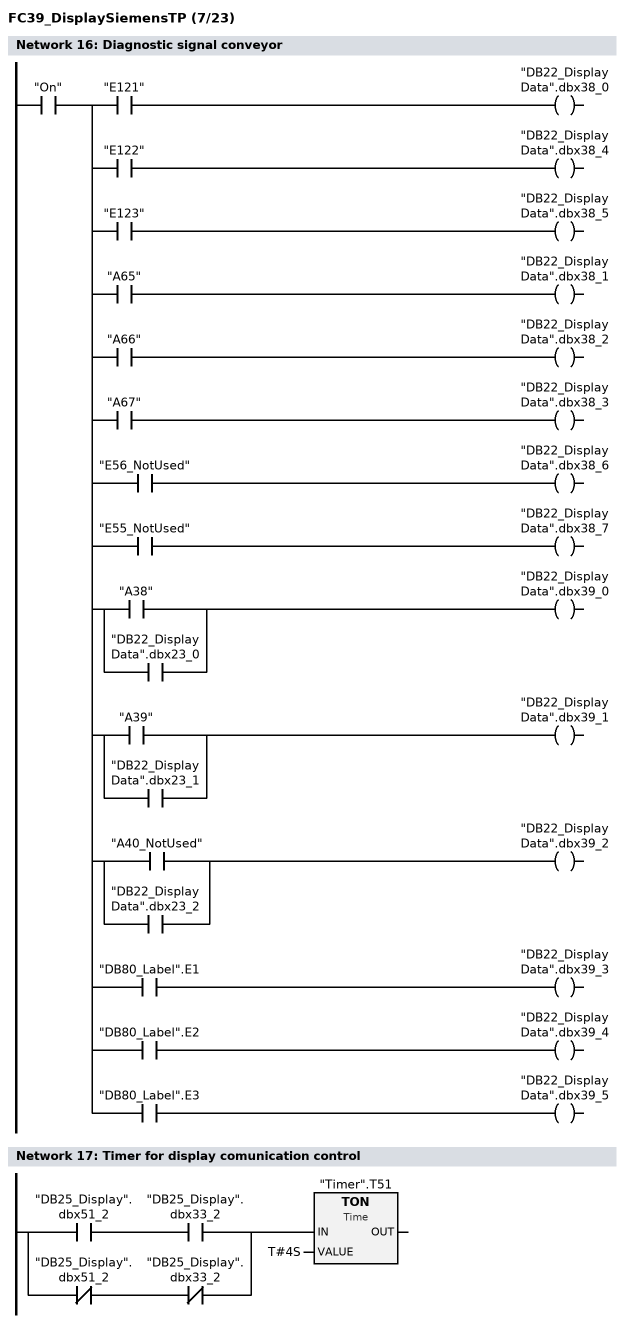
   RUNG wire#powerrail
      Contact( "On" )
      wire#w1
      Contact( "E121" )
      Coil( "DB22_DisplayData".dbx38_0 )
   END_RUNG
   RUNG wire#w1
      Contact( "E122" )
      Coil( "DB22_DisplayData".dbx38_4 )
   END_RUNG
   RUNG wire#w1
      Contact( "E123" )
      Coil( "DB22_DisplayData".dbx38_5 )
   END_RUNG
   RUNG wire#w1
      Contact( "A65" )
      Coil( "DB22_DisplayData".dbx38_1 )
   END_RUNG
   RUNG wire#w1
      Contact( "A66" )
      Coil( "DB22_DisplayData".dbx38_2 )
   END_RUNG
   RUNG wire#w1
      Contact( "A67" )
      Coil( "DB22_DisplayData".dbx38_3 )
   END_RUNG
   RUNG wire#w1
      Contact( "E56_NotUsed" )
      Coil( "DB22_DisplayData".dbx38_6 )
   END_RUNG
   RUNG wire#w1
      Contact( "E55_NotUsed" )
      Coil( "DB22_DisplayData".dbx38_7 )
   END_RUNG
   RUNG wire#w1
      Contact( "A38" )
      wire#w2
      Coil( "DB22_DisplayData".dbx39_0 )
   END_RUNG
   RUNG wire#w1
      Contact( "DB22_DisplayData".dbx23_0 )
   END_RUNG wire#w2
   RUNG wire#w1
      Contact( "A39" )
      wire#w3
      Coil( "DB22_DisplayData".dbx39_1 )
   END_RUNG
   RUNG wire#w1
      Contact( "DB22_DisplayData".dbx23_1 )
   END_RUNG wire#w3
   RUNG wire#w1
      Contact( "A40_NotUsed" )
      wire#w4
      Coil( "DB22_DisplayData".dbx39_2 )
   END_RUNG
   RUNG wire#w1
      Contact( "DB22_DisplayData".dbx23_2 )
   END_RUNG wire#w4
   RUNG wire#w1
      Contact( "DB80_Label".E1 )
      Coil( "DB22_DisplayData".dbx39_3 )
   END_RUNG
   RUNG wire#w1
      Contact( "DB80_Label".E2 )
      Coil( "DB22_DisplayData".dbx39_4 )
   END_RUNG
   RUNG wire#w1
      Contact( "DB80_Label".E3 )
      Coil( "DB22_DisplayData".dbx39_5 )
   END_RUNG
   // the same network as SCL:
   "DB22_DisplayData".dbx38_0 := "On" AND "E121";
   "DB22_DisplayData".dbx38_4 := "On" AND "E122";
   "DB22_DisplayData".dbx38_5 := "On" AND "E123";
   "DB22_DisplayData".dbx38_1 := "On" AND "A65";
   "DB22_DisplayData".dbx38_2 := "On" AND "A66";
   "DB22_DisplayData".dbx38_3 := "On" AND "A67";
   "DB22_DisplayData".dbx38_6 := "On" AND "E56_NotUsed";
   "DB22_DisplayData".dbx38_7 := "On" AND "E55_NotUsed";
   "DB22_DisplayData".dbx39_0 := "On" AND ("A38" OR "DB22_DisplayData".dbx23_0);
   "DB22_DisplayData".dbx39_1 := "On" AND ("A39" OR "DB22_DisplayData".dbx23_1);
   "DB22_DisplayData".dbx39_2 := "On" AND ("A40_NotUsed" OR "DB22_DisplayData".dbx23_2);
   "DB22_DisplayData".dbx39_3 := "On" AND "DB80_Label".E1;
   "DB22_DisplayData".dbx39_4 := "On" AND "DB80_Label".E2;
   "DB22_DisplayData".dbx39_5 := "On" AND "DB80_Label".E3;
END_REGION

REGION Network 17: Timer for display comunication control
   "Timer".T51.TON(IN := ("DB25_Display".dbx51_2 AND "DB25_Display".dbx33_2) OR (NOT "DB25_Display".dbx51_2 AND NOT "DB25_Display".dbx33_2), PT := T#4S);   // TON coil
END_REGION

REGION Network 18: Support for display communication timeout
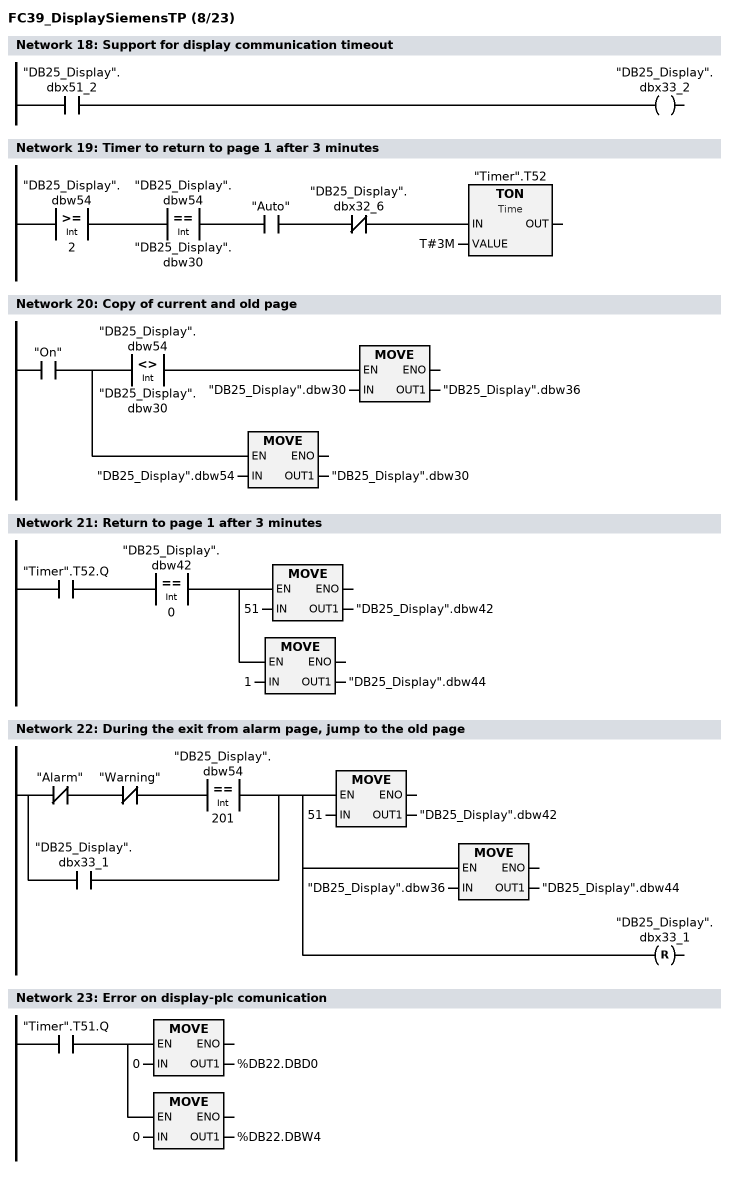
   RUNG wire#powerrail
      Contact( "DB25_Display".dbx51_2 )
      Coil( "DB25_Display".dbx33_2 )
   END_RUNG
   // the same network as SCL:
   "DB25_Display".dbx33_2 := "DB25_Display".dbx51_2;
END_REGION

REGION Network 19: Timer to return to page 1 after 3 minutes
   "Timer".T52.TON(IN := ("DB25_Display".dbw54 >= 2) AND ("DB25_Display".dbw54 = "DB25_Display".dbw30) AND "Auto" AND NOT "DB25_Display".dbx32_6, PT := T#3M);   // TON coil
END_REGION

REGION Network 20: Copy of current and old page
   RUNG wire#powerrail
      Contact( "On" )
      wire#w1
      { S7_Templates := "SrcType := Int" } NE_Contact(in1 := "DB25_Display".dbw54, in2 := "DB25_Display".dbw30)
      { S7_GenerateENO := "TRUE" } Move(in := "DB25_Display".dbw30, out1 => "DB25_Display".dbw36)
   END_RUNG
   RUNG wire#w1
      { S7_GenerateENO := "TRUE" } Move(in := "DB25_Display".dbw54, out1 => "DB25_Display".dbw30)
   END_RUNG
   // the same network as SCL:
   IF "On" AND ("DB25_Display".dbw54 <> "DB25_Display".dbw30) THEN
       "DB25_Display".dbw36 := "DB25_Display".dbw30;
   END_IF;
   IF "On" THEN "DB25_Display".dbw30 := "DB25_Display".dbw54; END_IF;
END_REGION

REGION Network 21: Return to page 1 after 3 minutes
   RUNG wire#powerrail
      Contact( "Timer".T52.Q )
      { S7_Templates := "SrcType := Int" } EQ_Contact(in1 := "DB25_Display".dbw42, in2 := 0)
      wire#w1
      { S7_GenerateENO := "TRUE" } Move(in := 51, out1 => "DB25_Display".dbw42)
   END_RUNG
   RUNG wire#w1
      { S7_GenerateENO := "TRUE" } Move(in := 1, out1 => "DB25_Display".dbw44)
   END_RUNG
   // the same network as SCL:
   #_w1 := "Timer".T52.Q AND ("DB25_Display".dbw42 = 0);
   IF #_w1 THEN
       "DB25_Display".dbw42 := 51;
       "DB25_Display".dbw44 := 1;
   END_IF;
END_REGION

REGION Network 22: During the exit from alarm page, jump to the old page
   RUNG wire#powerrail
      I_Contact( "Alarm" )
      I_Contact( "Warning" )
      { S7_Templates := "SrcType := Int" } EQ_Contact(in1 := "DB25_Display".dbw54, in2 := 201)
      wire#w1
      { S7_GenerateENO := "TRUE" } Move(in := 51, out1 => "DB25_Display".dbw42)
   END_RUNG
   RUNG wire#powerrail
      Contact( "DB25_Display".dbx33_1 )
   END_RUNG wire#w1
   RUNG wire#w1
      { S7_GenerateENO := "TRUE" } Move(in := "DB25_Display".dbw36, out1 => "DB25_Display".dbw44)
   END_RUNG
   RUNG wire#w1
      R_Coil( "DB25_Display".dbx33_1 )
   END_RUNG
   // the same network as SCL:
   IF (NOT "Alarm" AND NOT "Warning" AND ("DB25_Display".dbw54 = 201)) OR "DB25_Display".dbx33_1 THEN
       "DB25_Display".dbw42 := 51;
       "DB25_Display".dbw44 := "DB25_Display".dbw36;
       "DB25_Display".dbx33_1 := FALSE;
   END_IF;
END_REGION

REGION Network 23: Error on display-plc comunication
   RUNG wire#powerrail
      Contact( "Timer".T51.Q )
      wire#w1
      { S7_GenerateENO := "TRUE" } Move(in := 0, out1 => %DB22.DBD0)
   END_RUNG
   RUNG wire#w1
      { S7_GenerateENO := "TRUE" } Move(in := 0, out1 => %DB22.DBW4)
   END_RUNG
   // the same network as SCL:
   IF "Timer".T51.Q THEN
       %DB22.DBD0 := 0;
       %DB22.DBW4 := 0;
   END_IF;
END_REGION

REGION Network 24: Machine mode on Display
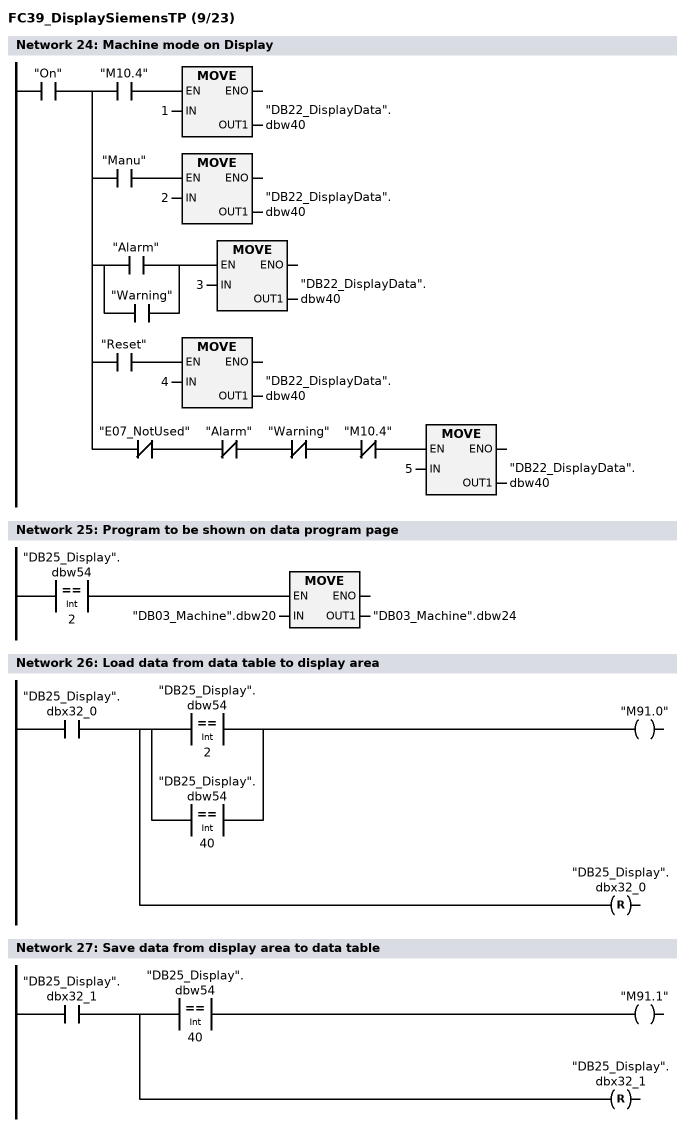
   RUNG wire#powerrail
      Contact( "On" )
      wire#w1
      Contact( "M10.4" )
      { S7_GenerateENO := "TRUE" } Move(in := 1, out1 => "DB22_DisplayData".dbw40)
   END_RUNG
   RUNG wire#w1
      Contact( "Manu" )
      { S7_GenerateENO := "TRUE" } Move(in := 2, out1 => "DB22_DisplayData".dbw40)
   END_RUNG
   RUNG wire#w1
      Contact( "Alarm" )
      wire#w2
      { S7_GenerateENO := "TRUE" } Move(in := 3, out1 => "DB22_DisplayData".dbw40)
   END_RUNG
   RUNG wire#w1
      Contact( "Warning" )
   END_RUNG wire#w2
   RUNG wire#w1
      Contact( "Reset" )
      { S7_GenerateENO := "TRUE" } Move(in := 4, out1 => "DB22_DisplayData".dbw40)
   END_RUNG
   RUNG wire#w1
      I_Contact( "E07_NotUsed" )
      I_Contact( "Alarm" )
      I_Contact( "Warning" )
      I_Contact( "M10.4" )
      { S7_GenerateENO := "TRUE" } Move(in := 5, out1 => "DB22_DisplayData".dbw40)
   END_RUNG
   // the same network as SCL:
   IF "On" AND "M10.4" THEN "DB22_DisplayData".dbw40 := 1; END_IF;
   IF "On" AND "Manu" THEN "DB22_DisplayData".dbw40 := 2; END_IF;
   IF "On" AND ("Alarm" OR "Warning") THEN "DB22_DisplayData".dbw40 := 3; END_IF;
   IF "On" AND "Reset" THEN "DB22_DisplayData".dbw40 := 4; END_IF;
   IF "On" AND NOT "E07_NotUsed" AND NOT "Alarm" AND NOT "Warning" AND NOT "M10.4" THEN
       "DB22_DisplayData".dbw40 := 5;
   END_IF;
END_REGION

REGION Network 25: Program to be shown on data program page
   RUNG wire#powerrail
      { S7_Templates := "SrcType := Int" } EQ_Contact(in1 := "DB25_Display".dbw54, in2 := 2)
      { S7_GenerateENO := "TRUE" } Move(in := "DB03_Machine".dbw20, out1 => "DB03_Machine".dbw24)
   END_RUNG
   // the same network as SCL:
   IF "DB25_Display".dbw54 = 2 THEN "DB03_Machine".dbw24 := "DB03_Machine".dbw20; END_IF;
END_REGION

REGION Network 26: Load data from data table to display area
   RUNG wire#powerrail
      Contact( "DB25_Display".dbx32_0 )
      wire#w1
      { S7_Templates := "SrcType := Int" } EQ_Contact(in1 := "DB25_Display".dbw54, in2 := 2)
      wire#w2
      Coil( "M91.0" )
   END_RUNG
   RUNG wire#w1
      { S7_Templates := "SrcType := Int" } EQ_Contact(in1 := "DB25_Display".dbw54, in2 := 40)
   END_RUNG wire#w2
   RUNG wire#w1
      R_Coil( "DB25_Display".dbx32_0 )
   END_RUNG
   // the same network as SCL:
   "M91.0" := "DB25_Display".dbx32_0 AND (("DB25_Display".dbw54 = 2) OR ("DB25_Display".dbw54 = 40));
   IF "DB25_Display".dbx32_0 THEN "DB25_Display".dbx32_0 := FALSE; END_IF;
END_REGION

REGION Network 27: Save data from display area to data table
   RUNG wire#powerrail
      Contact( "DB25_Display".dbx32_1 )
      wire#w1
      { S7_Templates := "SrcType := Int" } EQ_Contact(in1 := "DB25_Display".dbw54, in2 := 40)
      Coil( "M91.1" )
   END_RUNG
   RUNG wire#w1
      R_Coil( "DB25_Display".dbx32_1 )
   END_RUNG
   // the same network as SCL:
   "M91.1" := "DB25_Display".dbx32_1 AND ("DB25_Display".dbw54 = 40);
   IF "DB25_Display".dbx32_1 THEN "DB25_Display".dbx32_1 := FALSE; END_IF;
END_REGION

REGION Network 28: Program bit: Blink load button
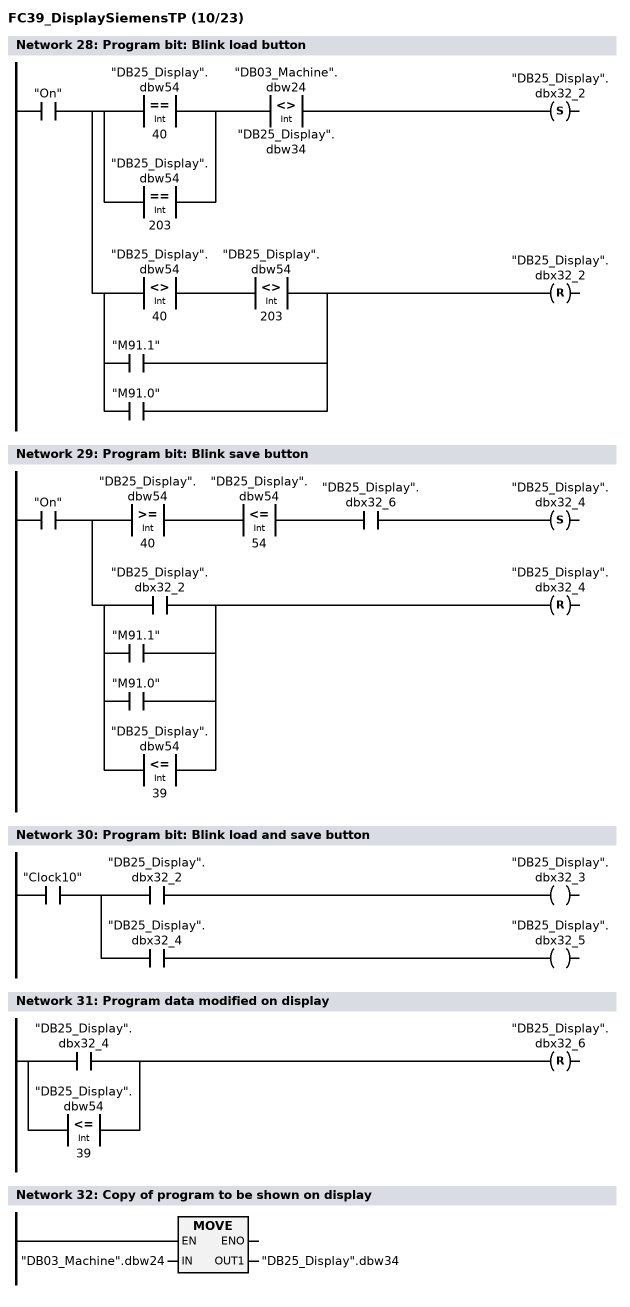
   RUNG wire#powerrail
      Contact( "On" )
      wire#w1
      { S7_Templates := "SrcType := Int" } EQ_Contact(in1 := "DB25_Display".dbw54, in2 := 40)
      wire#w2
      { S7_Templates := "SrcType := Int" } NE_Contact(in1 := "DB03_Machine".dbw24, in2 := "DB25_Display".dbw34)
      S_Coil( "DB25_Display".dbx32_2 )
   END_RUNG
   RUNG wire#w1
      { S7_Templates := "SrcType := Int" } EQ_Contact(in1 := "DB25_Display".dbw54, in2 := 203)
   END_RUNG wire#w2
   RUNG wire#w1
      { S7_Templates := "SrcType := Int" } NE_Contact(in1 := "DB25_Display".dbw54, in2 := 40)
      { S7_Templates := "SrcType := Int" } NE_Contact(in1 := "DB25_Display".dbw54, in2 := 203)
      wire#w3
      R_Coil( "DB25_Display".dbx32_2 )
   END_RUNG
   RUNG wire#w1
      Contact( "M91.1" )
   END_RUNG wire#w3
   RUNG wire#w1
      Contact( "M91.0" )
   END_RUNG wire#w3
   // the same network as SCL:
   IF "On" AND (("DB25_Display".dbw54 = 40) OR ("DB25_Display".dbw54 = 203)) AND ("DB03_Machine".dbw24 <> "DB25_Display".dbw34) THEN
       "DB25_Display".dbx32_2 := TRUE;
   END_IF;
   IF "On" AND ((("DB25_Display".dbw54 <> 40) AND ("DB25_Display".dbw54 <> 203)) OR "M91.1" OR "M91.0") THEN
       "DB25_Display".dbx32_2 := FALSE;
   END_IF;
END_REGION

REGION Network 29: Program bit: Blink save button
   RUNG wire#powerrail
      Contact( "On" )
      wire#w1
      { S7_Templates := "SrcType := Int" } GE_Contact(in1 := "DB25_Display".dbw54, in2 := 40)
      { S7_Templates := "SrcType := Int" } LE_Contact(in1 := "DB25_Display".dbw54, in2 := 54)
      Contact( "DB25_Display".dbx32_6 )
      S_Coil( "DB25_Display".dbx32_4 )
   END_RUNG
   RUNG wire#w1
      Contact( "DB25_Display".dbx32_2 )
      wire#w2
      R_Coil( "DB25_Display".dbx32_4 )
   END_RUNG
   RUNG wire#w1
      Contact( "M91.1" )
   END_RUNG wire#w2
   RUNG wire#w1
      Contact( "M91.0" )
   END_RUNG wire#w2
   RUNG wire#w1
      { S7_Templates := "SrcType := Int" } LE_Contact(in1 := "DB25_Display".dbw54, in2 := 39)
   END_RUNG wire#w2
   // the same network as SCL:
   IF "On" AND ("DB25_Display".dbw54 >= 40) AND ("DB25_Display".dbw54 <= 54) AND "DB25_Display".dbx32_6 THEN
       "DB25_Display".dbx32_4 := TRUE;
   END_IF;
   IF "On" AND ("DB25_Display".dbx32_2 OR "M91.1" OR "M91.0" OR ("DB25_Display".dbw54 <= 39)) THEN
       "DB25_Display".dbx32_4 := FALSE;
   END_IF;
END_REGION

REGION Network 30: Program bit: Blink load and save button
   RUNG wire#powerrail
      Contact( "Clock10" )
      wire#w1
      Contact( "DB25_Display".dbx32_2 )
      Coil( "DB25_Display".dbx32_3 )
   END_RUNG
   RUNG wire#w1
      Contact( "DB25_Display".dbx32_4 )
      Coil( "DB25_Display".dbx32_5 )
   END_RUNG
   // the same network as SCL:
   "DB25_Display".dbx32_3 := "Clock10" AND "DB25_Display".dbx32_2;
   "DB25_Display".dbx32_5 := "Clock10" AND "DB25_Display".dbx32_4;
END_REGION

REGION Network 31: Program data modified on display
   RUNG wire#powerrail
      Contact( "DB25_Display".dbx32_4 )
      wire#w1
      R_Coil( "DB25_Display".dbx32_6 )
   END_RUNG
   RUNG wire#powerrail
      { S7_Templates := "SrcType := Int" } LE_Contact(in1 := "DB25_Display".dbw54, in2 := 39)
   END_RUNG wire#w1
   // the same network as SCL:
   IF "DB25_Display".dbx32_4 OR ("DB25_Display".dbw54 <= 39) THEN "DB25_Display".dbx32_6 := FALSE; END_IF;
END_REGION

REGION Network 32: Copy of program to be shown on display
   RUNG wire#powerrail
      { S7_GenerateENO := "TRUE" } Move(in := "DB03_Machine".dbw24, out1 => "DB25_Display".dbw34)
   END_RUNG
   // the same network as SCL:
   "DB25_Display".dbw34 := "DB03_Machine".dbw24;
END_REGION

REGION Network 33: Grey bar data: Active program
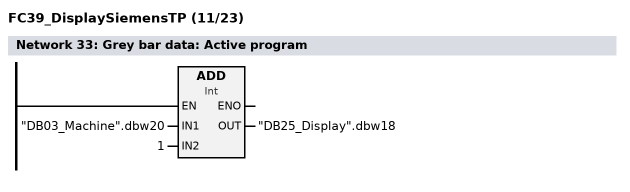
   RUNG wire#powerrail
      { S7_Templates := "SrcType := Int"; S7_GenerateENO := "TRUE" } Add(in1 := "DB03_Machine".dbw20, in2 := 1, out => "DB25_Display".dbw18)
   END_RUNG
   // the same network as SCL:
   "DB25_Display".dbw18 := "DB03_Machine".dbw20 + 1;
END_REGION

REGION Network 35: Support memory for pressure plate grey bar
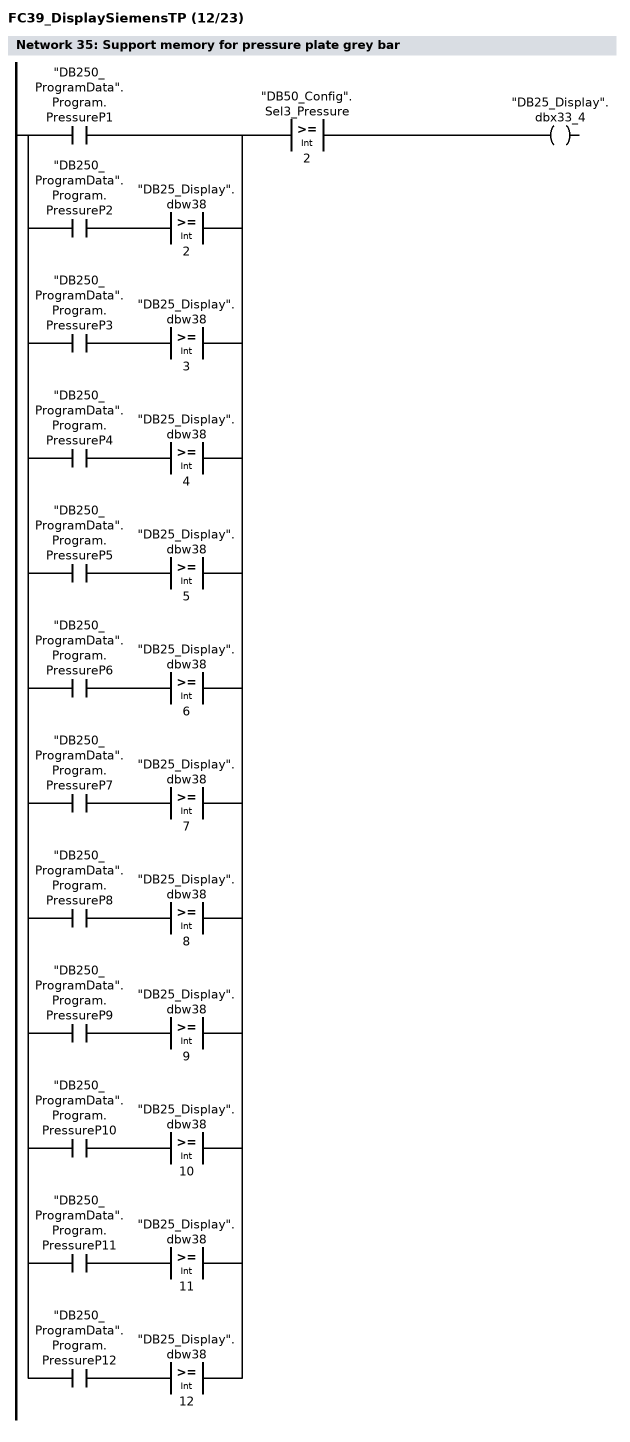
   RUNG wire#powerrail
      Contact( "DB250_ProgramData".Program.PressureP1 )
      wire#w1
      { S7_Templates := "SrcType := Int" } GE_Contact(in1 := "DB50_Config".Sel3_Pressure, in2 := 2)
      Coil( "DB25_Display".dbx33_4 )
   END_RUNG
   RUNG wire#powerrail
      Contact( "DB250_ProgramData".Program.PressureP2 )
      { S7_Templates := "SrcType := Int" } GE_Contact(in1 := "DB25_Display".dbw38, in2 := 2)
   END_RUNG wire#w1
   RUNG wire#powerrail
      Contact( "DB250_ProgramData".Program.PressureP3 )
      { S7_Templates := "SrcType := Int" } GE_Contact(in1 := "DB25_Display".dbw38, in2 := 3)
   END_RUNG wire#w1
   RUNG wire#powerrail
      Contact( "DB250_ProgramData".Program.PressureP4 )
      { S7_Templates := "SrcType := Int" } GE_Contact(in1 := "DB25_Display".dbw38, in2 := 4)
   END_RUNG wire#w1
   RUNG wire#powerrail
      Contact( "DB250_ProgramData".Program.PressureP5 )
      { S7_Templates := "SrcType := Int" } GE_Contact(in1 := "DB25_Display".dbw38, in2 := 5)
   END_RUNG wire#w1
   RUNG wire#powerrail
      Contact( "DB250_ProgramData".Program.PressureP6 )
      { S7_Templates := "SrcType := Int" } GE_Contact(in1 := "DB25_Display".dbw38, in2 := 6)
   END_RUNG wire#w1
   RUNG wire#powerrail
      Contact( "DB250_ProgramData".Program.PressureP7 )
      { S7_Templates := "SrcType := Int" } GE_Contact(in1 := "DB25_Display".dbw38, in2 := 7)
   END_RUNG wire#w1
   RUNG wire#powerrail
      Contact( "DB250_ProgramData".Program.PressureP8 )
      { S7_Templates := "SrcType := Int" } GE_Contact(in1 := "DB25_Display".dbw38, in2 := 8)
   END_RUNG wire#w1
   RUNG wire#powerrail
      Contact( "DB250_ProgramData".Program.PressureP9 )
      { S7_Templates := "SrcType := Int" } GE_Contact(in1 := "DB25_Display".dbw38, in2 := 9)
   END_RUNG wire#w1
   RUNG wire#powerrail
      Contact( "DB250_ProgramData".Program.PressureP10 )
      { S7_Templates := "SrcType := Int" } GE_Contact(in1 := "DB25_Display".dbw38, in2 := 10)
   END_RUNG wire#w1
   RUNG wire#powerrail
      Contact( "DB250_ProgramData".Program.PressureP11 )
      { S7_Templates := "SrcType := Int" } GE_Contact(in1 := "DB25_Display".dbw38, in2 := 11)
   END_RUNG wire#w1
   RUNG wire#powerrail
      Contact( "DB250_ProgramData".Program.PressureP12 )
      { S7_Templates := "SrcType := Int" } GE_Contact(in1 := "DB25_Display".dbw38, in2 := 12)
   END_RUNG wire#w1
   // the same network as SCL:
   "DB25_Display".dbx33_4 := ("DB250_ProgramData".Program.PressureP1 OR ("DB250_ProgramData".Program.PressureP2 AND ("DB25_Display".dbw38 >= 2)) OR ("DB250_ProgramData".Program.PressureP3 AND ("DB25_Display".dbw38 >= 3)) OR ("DB250_ProgramData".Program.PressureP4 AND ("DB25_Display".dbw38 >= 4)) OR ("DB250_ProgramData".Program.PressureP5 AND ("DB25_Display".dbw38 >= 5)) OR ("DB250_ProgramData".Program.PressureP6 AND ("DB25_Display".dbw38 >= 6)) OR ("DB250_ProgramData".Program.PressureP7 AND ("DB25_Display".dbw38 >= 7)) OR ("DB250_ProgramData".Program.PressureP8 AND ("DB25_Display".dbw38 >= 8)) OR ("DB250_ProgramData".Program.PressureP9 AND ("DB25_Display".dbw38 >= 9)) OR ("DB250_ProgramData".Program.PressureP10 AND ("DB25_Display".dbw38 >= 10)) OR ("DB250_ProgramData".Program.PressureP11 AND ("DB25_Display".dbw38 >= 11)) OR ("DB250_ProgramData".Program.PressureP12 AND ("DB25_Display".dbw38 >= 12))) AND ("DB50_Config".Sel3_Pressure >= 2);
END_REGION

REGION Network 36: Support memory for lifter grey bar
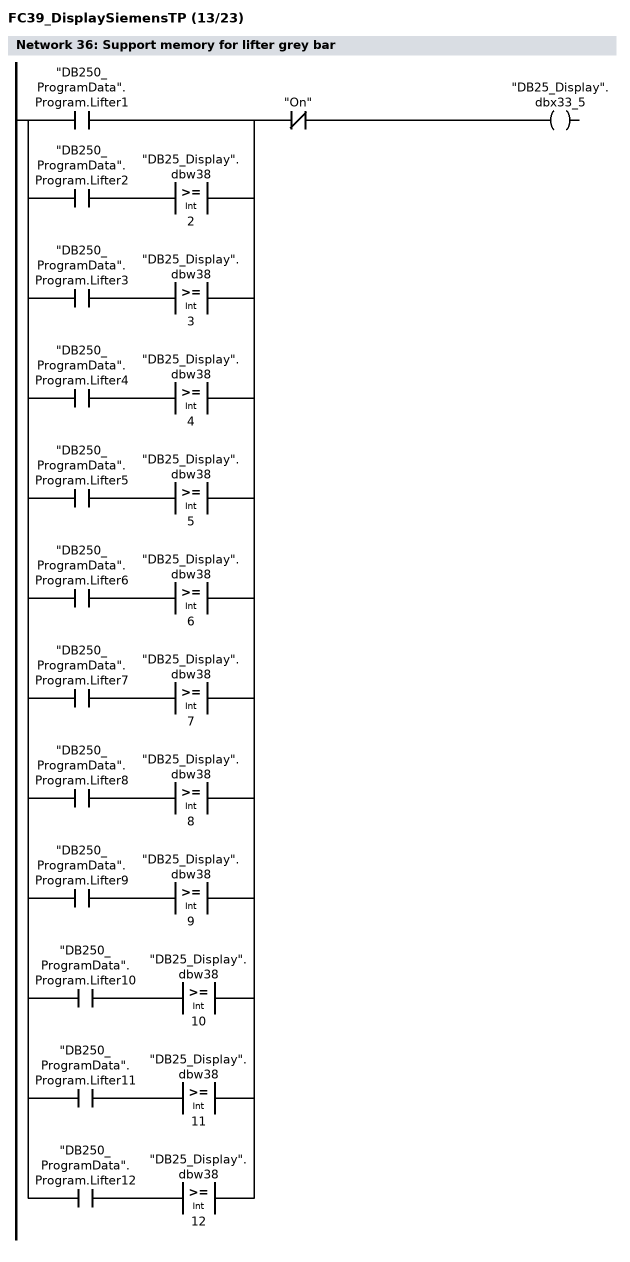
   RUNG wire#powerrail
      Contact( "DB250_ProgramData".Program.Lifter1 )
      wire#w1
      I_Contact( "On" )
      Coil( "DB25_Display".dbx33_5 )
   END_RUNG
   RUNG wire#powerrail
      Contact( "DB250_ProgramData".Program.Lifter2 )
      { S7_Templates := "SrcType := Int" } GE_Contact(in1 := "DB25_Display".dbw38, in2 := 2)
   END_RUNG wire#w1
   RUNG wire#powerrail
      Contact( "DB250_ProgramData".Program.Lifter3 )
      { S7_Templates := "SrcType := Int" } GE_Contact(in1 := "DB25_Display".dbw38, in2 := 3)
   END_RUNG wire#w1
   RUNG wire#powerrail
      Contact( "DB250_ProgramData".Program.Lifter4 )
      { S7_Templates := "SrcType := Int" } GE_Contact(in1 := "DB25_Display".dbw38, in2 := 4)
   END_RUNG wire#w1
   RUNG wire#powerrail
      Contact( "DB250_ProgramData".Program.Lifter5 )
      { S7_Templates := "SrcType := Int" } GE_Contact(in1 := "DB25_Display".dbw38, in2 := 5)
   END_RUNG wire#w1
   RUNG wire#powerrail
      Contact( "DB250_ProgramData".Program.Lifter6 )
      { S7_Templates := "SrcType := Int" } GE_Contact(in1 := "DB25_Display".dbw38, in2 := 6)
   END_RUNG wire#w1
   RUNG wire#powerrail
      Contact( "DB250_ProgramData".Program.Lifter7 )
      { S7_Templates := "SrcType := Int" } GE_Contact(in1 := "DB25_Display".dbw38, in2 := 7)
   END_RUNG wire#w1
   RUNG wire#powerrail
      Contact( "DB250_ProgramData".Program.Lifter8 )
      { S7_Templates := "SrcType := Int" } GE_Contact(in1 := "DB25_Display".dbw38, in2 := 8)
   END_RUNG wire#w1
   RUNG wire#powerrail
      Contact( "DB250_ProgramData".Program.Lifter9 )
      { S7_Templates := "SrcType := Int" } GE_Contact(in1 := "DB25_Display".dbw38, in2 := 9)
   END_RUNG wire#w1
   RUNG wire#powerrail
      Contact( "DB250_ProgramData".Program.Lifter10 )
      { S7_Templates := "SrcType := Int" } GE_Contact(in1 := "DB25_Display".dbw38, in2 := 10)
   END_RUNG wire#w1
   RUNG wire#powerrail
      Contact( "DB250_ProgramData".Program.Lifter11 )
      { S7_Templates := "SrcType := Int" } GE_Contact(in1 := "DB25_Display".dbw38, in2 := 11)
   END_RUNG wire#w1
   RUNG wire#powerrail
      Contact( "DB250_ProgramData".Program.Lifter12 )
      { S7_Templates := "SrcType := Int" } GE_Contact(in1 := "DB25_Display".dbw38, in2 := 12)
   END_RUNG wire#w1
   // the same network as SCL:
   "DB25_Display".dbx33_5 := ("DB250_ProgramData".Program.Lifter1 OR ("DB250_ProgramData".Program.Lifter2 AND ("DB25_Display".dbw38 >= 2)) OR ("DB250_ProgramData".Program.Lifter3 AND ("DB25_Display".dbw38 >= 3)) OR ("DB250_ProgramData".Program.Lifter4 AND ("DB25_Display".dbw38 >= 4)) OR ("DB250_ProgramData".Program.Lifter5 AND ("DB25_Display".dbw38 >= 5)) OR ("DB250_ProgramData".Program.Lifter6 AND ("DB25_Display".dbw38 >= 6)) OR ("DB250_ProgramData".Program.Lifter7 AND ("DB25_Display".dbw38 >= 7)) OR ("DB250_ProgramData".Program.Lifter8 AND ("DB25_Display".dbw38 >= 8)) OR ("DB250_ProgramData".Program.Lifter9 AND ("DB25_Display".dbw38 >= 9)) OR ("DB250_ProgramData".Program.Lifter10 AND ("DB25_Display".dbw38 >= 10)) OR ("DB250_ProgramData".Program.Lifter11 AND ("DB25_Display".dbw38 >= 11)) OR ("DB250_ProgramData".Program.Lifter12 AND ("DB25_Display".dbw38 >= 12))) AND NOT "On";
END_REGION

REGION Network 37: Grey bar data: Wrapping, Top, Pressure plate and Lifter
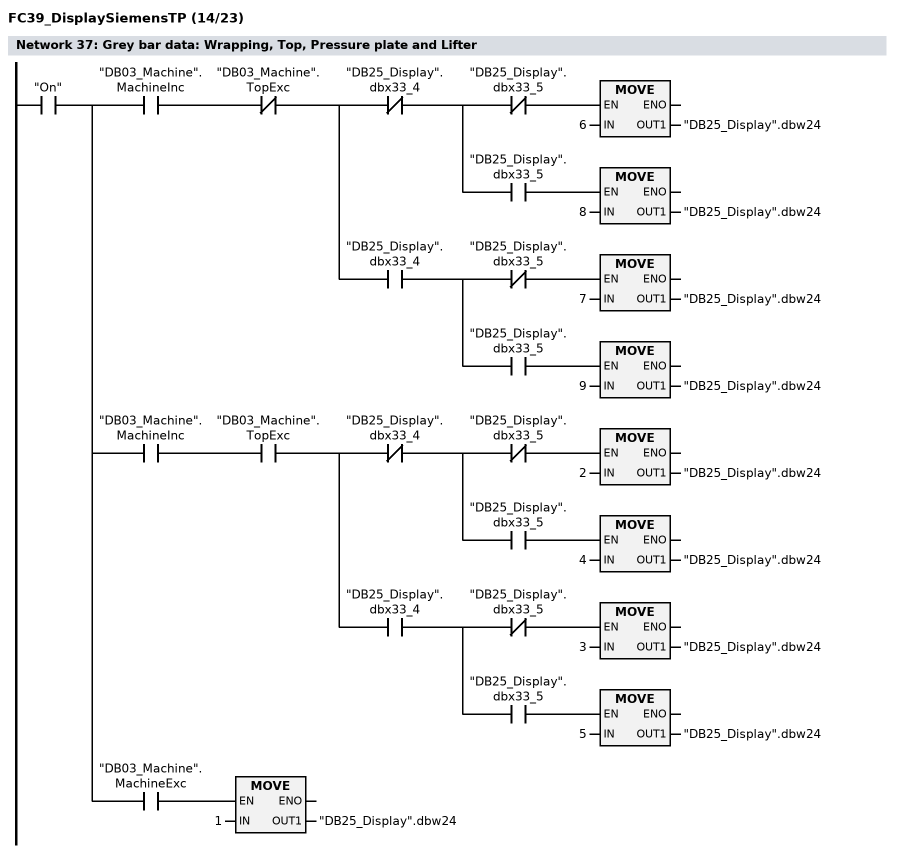
   RUNG wire#powerrail
      Contact( "On" )
      wire#w1
      Contact( "DB03_Machine".MachineInc )
      I_Contact( "DB03_Machine".TopExc )
      wire#w2
      I_Contact( "DB25_Display".dbx33_4 )
      wire#w3
      I_Contact( "DB25_Display".dbx33_5 )
      { S7_GenerateENO := "TRUE" } Move(in := 6, out1 => "DB25_Display".dbw24)
   END_RUNG
   RUNG wire#w3
      Contact( "DB25_Display".dbx33_5 )
      { S7_GenerateENO := "TRUE" } Move(in := 8, out1 => "DB25_Display".dbw24)
   END_RUNG
   RUNG wire#w2
      Contact( "DB25_Display".dbx33_4 )
      wire#w4
      I_Contact( "DB25_Display".dbx33_5 )
      { S7_GenerateENO := "TRUE" } Move(in := 7, out1 => "DB25_Display".dbw24)
   END_RUNG
   RUNG wire#w4
      Contact( "DB25_Display".dbx33_5 )
      { S7_GenerateENO := "TRUE" } Move(in := 9, out1 => "DB25_Display".dbw24)
   END_RUNG
   RUNG wire#w1
      Contact( "DB03_Machine".MachineInc )
      Contact( "DB03_Machine".TopExc )
      wire#w5
      I_Contact( "DB25_Display".dbx33_4 )
      wire#w6
      I_Contact( "DB25_Display".dbx33_5 )
      { S7_GenerateENO := "TRUE" } Move(in := 2, out1 => "DB25_Display".dbw24)
   END_RUNG
   RUNG wire#w6
      Contact( "DB25_Display".dbx33_5 )
      { S7_GenerateENO := "TRUE" } Move(in := 4, out1 => "DB25_Display".dbw24)
   END_RUNG
   RUNG wire#w5
      Contact( "DB25_Display".dbx33_4 )
      wire#w7
      I_Contact( "DB25_Display".dbx33_5 )
      { S7_GenerateENO := "TRUE" } Move(in := 3, out1 => "DB25_Display".dbw24)
   END_RUNG
   RUNG wire#w7
      Contact( "DB25_Display".dbx33_5 )
      { S7_GenerateENO := "TRUE" } Move(in := 5, out1 => "DB25_Display".dbw24)
   END_RUNG
   RUNG wire#w1
      Contact( "DB03_Machine".MachineExc )
      { S7_GenerateENO := "TRUE" } Move(in := 1, out1 => "DB25_Display".dbw24)
   END_RUNG
   // the same network as SCL:
   #_w1 := "On" AND "DB03_Machine".MachineInc AND NOT "DB03_Machine".TopExc;
   #_w2 := #_w1 AND NOT "DB25_Display".dbx33_4;
   IF #_w2 AND NOT "DB25_Display".dbx33_5 THEN "DB25_Display".dbw24 := 6; END_IF;
   IF #_w2 AND "DB25_Display".dbx33_5 THEN "DB25_Display".dbw24 := 8; END_IF;
   #_w3 := #_w1 AND "DB25_Display".dbx33_4;
   IF #_w3 AND NOT "DB25_Display".dbx33_5 THEN "DB25_Display".dbw24 := 7; END_IF;
   IF #_w3 AND "DB25_Display".dbx33_5 THEN "DB25_Display".dbw24 := 9; END_IF;
   #_w4 := "On" AND "DB03_Machine".MachineInc AND "DB03_Machine".TopExc;
   #_w5 := #_w4 AND NOT "DB25_Display".dbx33_4;
   IF #_w5 AND NOT "DB25_Display".dbx33_5 THEN "DB25_Display".dbw24 := 2; END_IF;
   IF #_w5 AND "DB25_Display".dbx33_5 THEN "DB25_Display".dbw24 := 4; END_IF;
   #_w6 := #_w4 AND "DB25_Display".dbx33_4;
   IF #_w6 AND NOT "DB25_Display".dbx33_5 THEN "DB25_Display".dbw24 := 3; END_IF;
   IF #_w6 AND "DB25_Display".dbx33_5 THEN "DB25_Display".dbw24 := 5; END_IF;
   IF "On" AND "DB03_Machine".MachineExc THEN "DB25_Display".dbw24 := 1; END_IF;
END_REGION

REGION Network 38: Grey bar data: Quote active
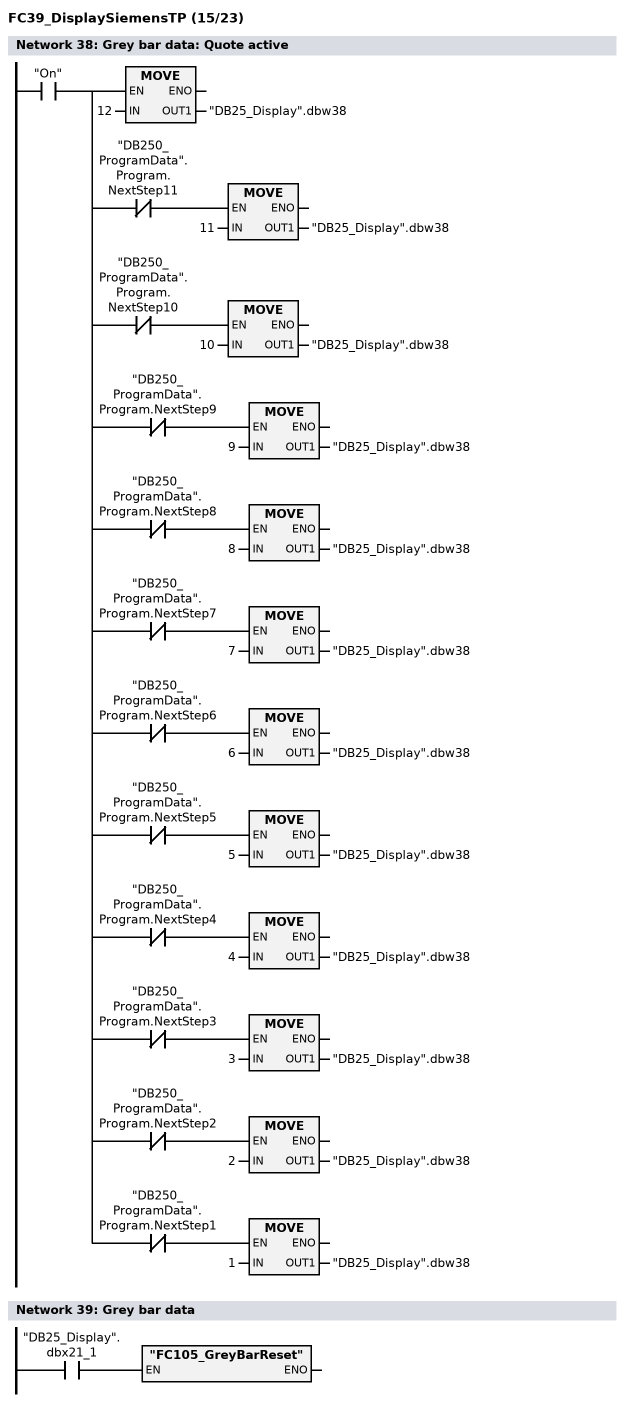
   RUNG wire#powerrail
      Contact( "On" )
      wire#w1
      { S7_GenerateENO := "TRUE" } Move(in := 12, out1 => "DB25_Display".dbw38)
   END_RUNG
   RUNG wire#w1
      I_Contact( "DB250_ProgramData".Program.NextStep11 )
      { S7_GenerateENO := "TRUE" } Move(in := 11, out1 => "DB25_Display".dbw38)
   END_RUNG
   RUNG wire#w1
      I_Contact( "DB250_ProgramData".Program.NextStep10 )
      { S7_GenerateENO := "TRUE" } Move(in := 10, out1 => "DB25_Display".dbw38)
   END_RUNG
   RUNG wire#w1
      I_Contact( "DB250_ProgramData".Program.NextStep9 )
      { S7_GenerateENO := "TRUE" } Move(in := 9, out1 => "DB25_Display".dbw38)
   END_RUNG
   RUNG wire#w1
      I_Contact( "DB250_ProgramData".Program.NextStep8 )
      { S7_GenerateENO := "TRUE" } Move(in := 8, out1 => "DB25_Display".dbw38)
   END_RUNG
   RUNG wire#w1
      I_Contact( "DB250_ProgramData".Program.NextStep7 )
      { S7_GenerateENO := "TRUE" } Move(in := 7, out1 => "DB25_Display".dbw38)
   END_RUNG
   RUNG wire#w1
      I_Contact( "DB250_ProgramData".Program.NextStep6 )
      { S7_GenerateENO := "TRUE" } Move(in := 6, out1 => "DB25_Display".dbw38)
   END_RUNG
   RUNG wire#w1
      I_Contact( "DB250_ProgramData".Program.NextStep5 )
      { S7_GenerateENO := "TRUE" } Move(in := 5, out1 => "DB25_Display".dbw38)
   END_RUNG
   RUNG wire#w1
      I_Contact( "DB250_ProgramData".Program.NextStep4 )
      { S7_GenerateENO := "TRUE" } Move(in := 4, out1 => "DB25_Display".dbw38)
   END_RUNG
   RUNG wire#w1
      I_Contact( "DB250_ProgramData".Program.NextStep3 )
      { S7_GenerateENO := "TRUE" } Move(in := 3, out1 => "DB25_Display".dbw38)
   END_RUNG
   RUNG wire#w1
      I_Contact( "DB250_ProgramData".Program.NextStep2 )
      { S7_GenerateENO := "TRUE" } Move(in := 2, out1 => "DB25_Display".dbw38)
   END_RUNG
   RUNG wire#w1
      I_Contact( "DB250_ProgramData".Program.NextStep1 )
      { S7_GenerateENO := "TRUE" } Move(in := 1, out1 => "DB25_Display".dbw38)
   END_RUNG
   // the same network as SCL:
   IF "On" THEN "DB25_Display".dbw38 := 12; END_IF;
   IF "On" AND NOT "DB250_ProgramData".Program.NextStep11 THEN "DB25_Display".dbw38 := 11; END_IF;
   IF "On" AND NOT "DB250_ProgramData".Program.NextStep10 THEN "DB25_Display".dbw38 := 10; END_IF;
   IF "On" AND NOT "DB250_ProgramData".Program.NextStep9 THEN "DB25_Display".dbw38 := 9; END_IF;
   IF "On" AND NOT "DB250_ProgramData".Program.NextStep8 THEN "DB25_Display".dbw38 := 8; END_IF;
   IF "On" AND NOT "DB250_ProgramData".Program.NextStep7 THEN "DB25_Display".dbw38 := 7; END_IF;
   IF "On" AND NOT "DB250_ProgramData".Program.NextStep6 THEN "DB25_Display".dbw38 := 6; END_IF;
   IF "On" AND NOT "DB250_ProgramData".Program.NextStep5 THEN "DB25_Display".dbw38 := 5; END_IF;
   IF "On" AND NOT "DB250_ProgramData".Program.NextStep4 THEN "DB25_Display".dbw38 := 4; END_IF;
   IF "On" AND NOT "DB250_ProgramData".Program.NextStep3 THEN "DB25_Display".dbw38 := 3; END_IF;
   IF "On" AND NOT "DB250_ProgramData".Program.NextStep2 THEN "DB25_Display".dbw38 := 2; END_IF;
   IF "On" AND NOT "DB250_ProgramData".Program.NextStep1 THEN "DB25_Display".dbw38 := 1; END_IF;
END_REGION

REGION Network 39: Grey bar data
   RUNG wire#powerrail
      Contact( "DB25_Display".dbx21_1 )
      "FC105_GreyBarReset"()
   END_RUNG
   // the same network as SCL:
   IF "DB25_Display".dbx21_1 THEN "FC105_GreyBarReset"(); END_IF;
END_REGION

REGION Network 40: Grey bar data
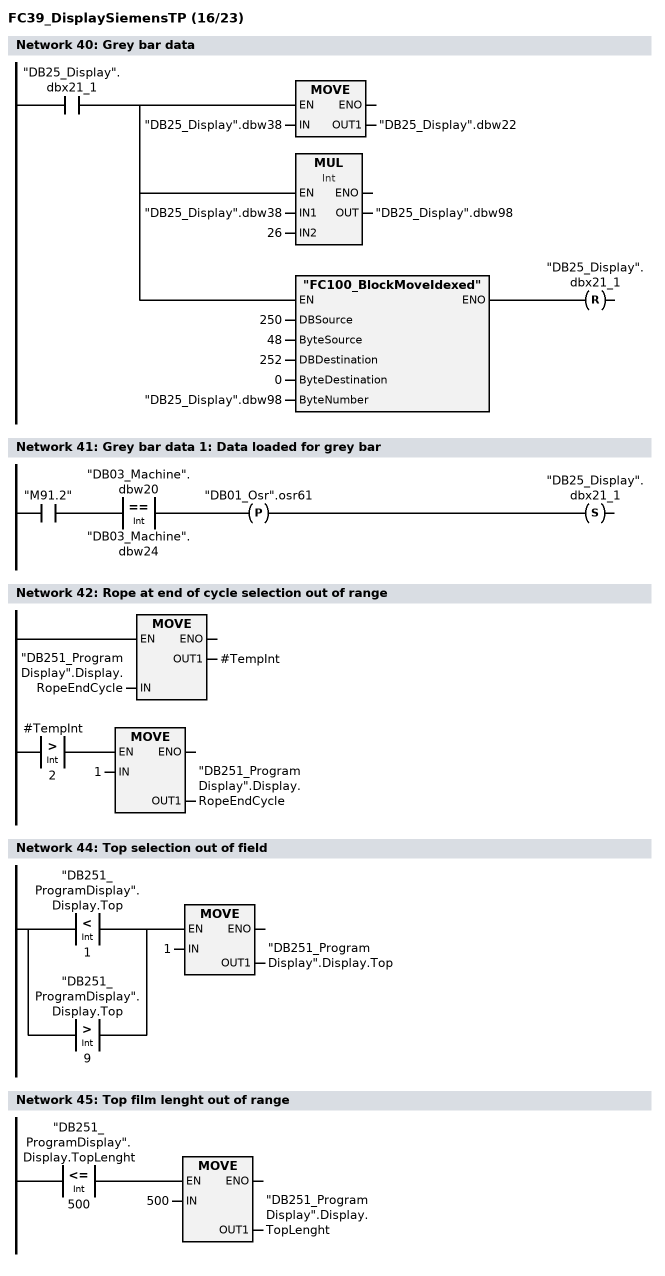
   RUNG wire#powerrail
      Contact( "DB25_Display".dbx21_1 )
      wire#w1
      { S7_GenerateENO := "TRUE" } Move(in := "DB25_Display".dbw38, out1 => "DB25_Display".dbw22)
   END_RUNG
   RUNG wire#w1
      { S7_Templates := "SrcType := Int"; S7_GenerateENO := "TRUE" } Mul(in1 := "DB25_Display".dbw38, in2 := 26, out => "DB25_Display".dbw98)
   END_RUNG
   RUNG wire#w1
      "FC100_BlockMoveIdexed"(DBSource := 250, ByteSource := 48, DBDestination := 252, ByteDestination := 0, ByteNumber := "DB25_Display".dbw98)
      R_Coil( "DB25_Display".dbx21_1 )
   END_RUNG
   // the same network as SCL:
   IF "DB25_Display".dbx21_1 THEN
       "DB25_Display".dbw22 := "DB25_Display".dbw38;
       "DB25_Display".dbw98 := "DB25_Display".dbw38 * 26;
   END_IF;
   "FC100_BlockMoveIdexed"(EN := "DB25_Display".dbx21_1,
                           DBSource := 250,
                           ByteSource := 48,
                           DBDestination := 252,
                           ByteDestination := 0,
                           ByteNumber := "DB25_Display".dbw98,
                           ENO => #_w1);
   IF #_w1 THEN "DB25_Display".dbx21_1 := FALSE; END_IF;
END_REGION

REGION Network 41: Grey bar data 1: Data loaded for grey bar
   RUNG wire#powerrail
      Contact( "M91.2" )
      { S7_Templates := "SrcType := Int" } EQ_Contact(in1 := "DB03_Machine".dbw20, in2 := "DB03_Machine".dbw24)
      P_Trig( "DB01_Osr".osr61 )
      S_Coil( "DB25_Display".dbx21_1 )
   END_RUNG
   // the same network as SCL:
   #_w1 := "M91.2" AND ("DB03_Machine".dbw20 = "DB03_Machine".dbw24);
   #_w2 := #_w1 AND NOT "DB01_Osr".osr61;   // rising edge
   "DB01_Osr".osr61 := #_w1;
   IF #_w2 THEN "DB25_Display".dbx21_1 := TRUE; END_IF;
END_REGION

REGION Network 42: Rope at end of cycle selection out of range
   RUNG wire#powerrail
      { S7_GenerateENO := "TRUE" } Move(in := "DB251_ProgramDisplay".Display.RopeEndCycle, out1 => #TempInt)
   END_RUNG
   RUNG wire#powerrail
      { S7_Templates := "SrcType := Int" } GT_Contact(in1 := #TempInt, in2 := 2)
      { S7_GenerateENO := "TRUE" } Move(in := 1, out1 => "DB251_ProgramDisplay".Display.RopeEndCycle)
   END_RUNG
   // the same network as SCL:
   #TempInt := "DB251_ProgramDisplay".Display.RopeEndCycle;
   IF #TempInt > 2 THEN "DB251_ProgramDisplay".Display.RopeEndCycle := 1; END_IF;
END_REGION

REGION Network 44: Top selection out of field
   RUNG wire#powerrail
      { S7_Templates := "SrcType := Int" } LT_Contact(in1 := "DB251_ProgramDisplay".Display.Top, in2 := 1)
      wire#w1
      { S7_GenerateENO := "TRUE" } Move(in := 1, out1 => "DB251_ProgramDisplay".Display.Top)
   END_RUNG
   RUNG wire#powerrail
      { S7_Templates := "SrcType := Int" } GT_Contact(in1 := "DB251_ProgramDisplay".Display.Top, in2 := 9)
   END_RUNG wire#w1
   // the same network as SCL:
   IF ("DB251_ProgramDisplay".Display.Top < 1) OR ("DB251_ProgramDisplay".Display.Top > 9) THEN
       "DB251_ProgramDisplay".Display.Top := 1;
   END_IF;
END_REGION

REGION Network 45: Top film lenght out of range
   RUNG wire#powerrail
      { S7_Templates := "SrcType := Int" } LE_Contact(in1 := "DB251_ProgramDisplay".Display.TopLenght, in2 := 500)
      { S7_GenerateENO := "TRUE" } Move(in := 500, out1 => "DB251_ProgramDisplay".Display.TopLenght)
   END_RUNG
   // the same network as SCL:
   IF "DB251_ProgramDisplay".Display.TopLenght <= 500 THEN
       "DB251_ProgramDisplay".Display.TopLenght := 500;
   END_IF;
END_REGION

REGION Network 46: Band unit out of range (1-6)
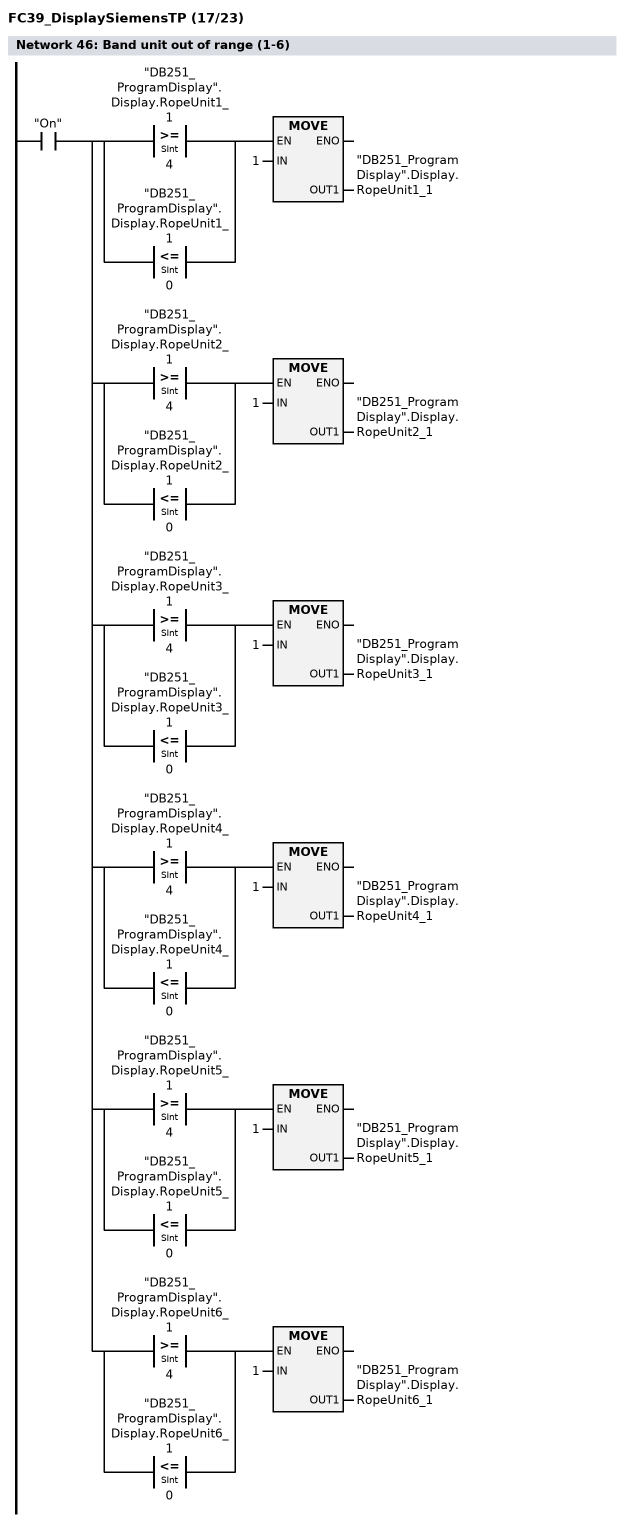
   RUNG wire#powerrail
      Contact( "On" )
      wire#w1
      { S7_Templates := "SrcType := SInt" } GE_Contact(in1 := "DB251_ProgramDisplay".Display.RopeUnit1_1, in2 := 4)
      wire#w2
      { S7_GenerateENO := "TRUE" } Move(in := 1, out1 => "DB251_ProgramDisplay".Display.RopeUnit1_1)
   END_RUNG
   RUNG wire#w1
      { S7_Templates := "SrcType := SInt" } LE_Contact(in1 := "DB251_ProgramDisplay".Display.RopeUnit1_1, in2 := 0)
   END_RUNG wire#w2
   RUNG wire#w1
      { S7_Templates := "SrcType := SInt" } GE_Contact(in1 := "DB251_ProgramDisplay".Display.RopeUnit2_1, in2 := 4)
      wire#w3
      { S7_GenerateENO := "TRUE" } Move(in := 1, out1 => "DB251_ProgramDisplay".Display.RopeUnit2_1)
   END_RUNG
   RUNG wire#w1
      { S7_Templates := "SrcType := SInt" } LE_Contact(in1 := "DB251_ProgramDisplay".Display.RopeUnit2_1, in2 := 0)
   END_RUNG wire#w3
   RUNG wire#w1
      { S7_Templates := "SrcType := SInt" } GE_Contact(in1 := "DB251_ProgramDisplay".Display.RopeUnit3_1, in2 := 4)
      wire#w4
      { S7_GenerateENO := "TRUE" } Move(in := 1, out1 => "DB251_ProgramDisplay".Display.RopeUnit3_1)
   END_RUNG
   RUNG wire#w1
      { S7_Templates := "SrcType := SInt" } LE_Contact(in1 := "DB251_ProgramDisplay".Display.RopeUnit3_1, in2 := 0)
   END_RUNG wire#w4
   RUNG wire#w1
      { S7_Templates := "SrcType := SInt" } GE_Contact(in1 := "DB251_ProgramDisplay".Display.RopeUnit4_1, in2 := 4)
      wire#w5
      { S7_GenerateENO := "TRUE" } Move(in := 1, out1 => "DB251_ProgramDisplay".Display.RopeUnit4_1)
   END_RUNG
   RUNG wire#w1
      { S7_Templates := "SrcType := SInt" } LE_Contact(in1 := "DB251_ProgramDisplay".Display.RopeUnit4_1, in2 := 0)
   END_RUNG wire#w5
   RUNG wire#w1
      { S7_Templates := "SrcType := SInt" } GE_Contact(in1 := "DB251_ProgramDisplay".Display.RopeUnit5_1, in2 := 4)
      wire#w6
      { S7_GenerateENO := "TRUE" } Move(in := 1, out1 => "DB251_ProgramDisplay".Display.RopeUnit5_1)
   END_RUNG
   RUNG wire#w1
      { S7_Templates := "SrcType := SInt" } LE_Contact(in1 := "DB251_ProgramDisplay".Display.RopeUnit5_1, in2 := 0)
   END_RUNG wire#w6
   RUNG wire#w1
      { S7_Templates := "SrcType := SInt" } GE_Contact(in1 := "DB251_ProgramDisplay".Display.RopeUnit6_1, in2 := 4)
      wire#w7
      { S7_GenerateENO := "TRUE" } Move(in := 1, out1 => "DB251_ProgramDisplay".Display.RopeUnit6_1)
   END_RUNG
   RUNG wire#w1
      { S7_Templates := "SrcType := SInt" } LE_Contact(in1 := "DB251_ProgramDisplay".Display.RopeUnit6_1, in2 := 0)
   END_RUNG wire#w7
   // the same network as SCL:
   IF "On" AND (("DB251_ProgramDisplay".Display.RopeUnit1_1 >= 4) OR ("DB251_ProgramDisplay".Display.RopeUnit1_1 <= 0)) THEN
       "DB251_ProgramDisplay".Display.RopeUnit1_1 := 1;
   END_IF;
   IF "On" AND (("DB251_ProgramDisplay".Display.RopeUnit2_1 >= 4) OR ("DB251_ProgramDisplay".Display.RopeUnit2_1 <= 0)) THEN
       "DB251_ProgramDisplay".Display.RopeUnit2_1 := 1;
   END_IF;
   IF "On" AND (("DB251_ProgramDisplay".Display.RopeUnit3_1 >= 4) OR ("DB251_ProgramDisplay".Display.RopeUnit3_1 <= 0)) THEN
       "DB251_ProgramDisplay".Display.RopeUnit3_1 := 1;
   END_IF;
   IF "On" AND (("DB251_ProgramDisplay".Display.RopeUnit4_1 >= 4) OR ("DB251_ProgramDisplay".Display.RopeUnit4_1 <= 0)) THEN
       "DB251_ProgramDisplay".Display.RopeUnit4_1 := 1;
   END_IF;
   IF "On" AND (("DB251_ProgramDisplay".Display.RopeUnit5_1 >= 4) OR ("DB251_ProgramDisplay".Display.RopeUnit5_1 <= 0)) THEN
       "DB251_ProgramDisplay".Display.RopeUnit5_1 := 1;
   END_IF;
   IF "On" AND (("DB251_ProgramDisplay".Display.RopeUnit6_1 >= 4) OR ("DB251_ProgramDisplay".Display.RopeUnit6_1 <= 0)) THEN
       "DB251_ProgramDisplay".Display.RopeUnit6_1 := 1;
   END_IF;
END_REGION

REGION Network 47: Band unit out of range (7-12)
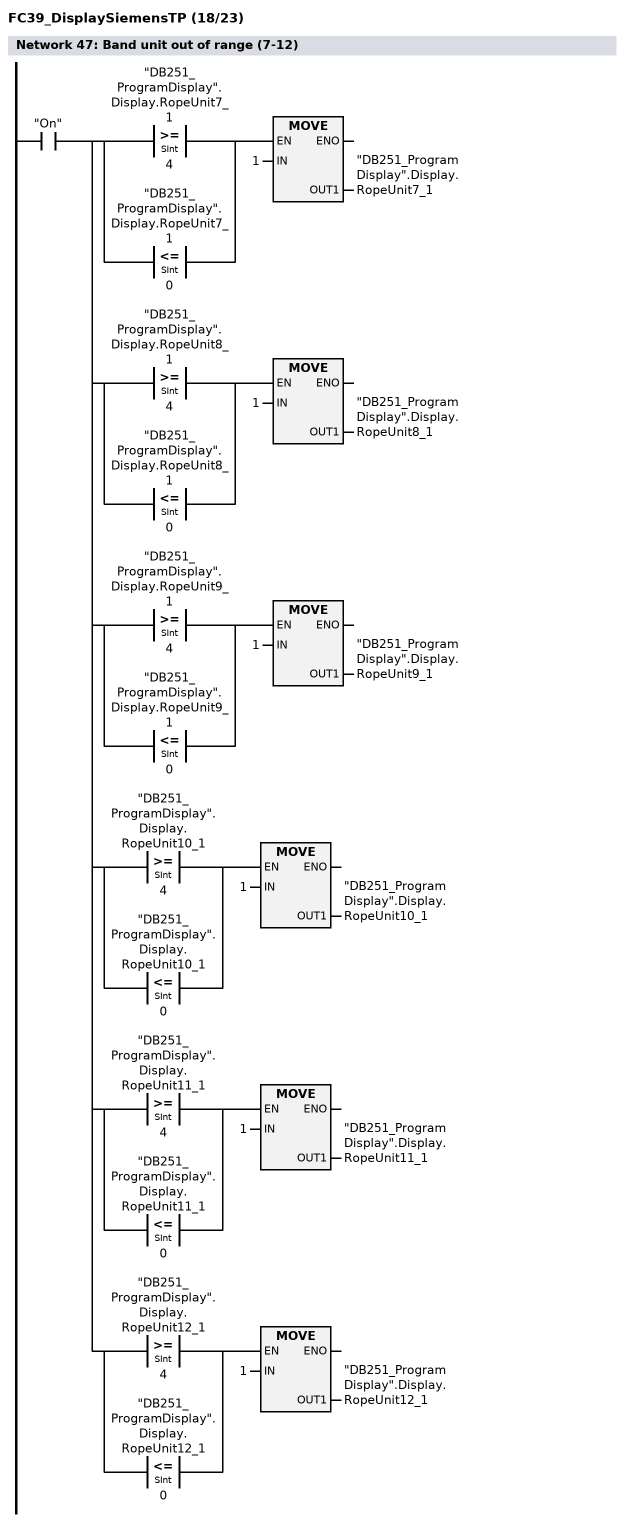
   RUNG wire#powerrail
      Contact( "On" )
      wire#w1
      { S7_Templates := "SrcType := SInt" } GE_Contact(in1 := "DB251_ProgramDisplay".Display.RopeUnit7_1, in2 := 4)
      wire#w2
      { S7_GenerateENO := "TRUE" } Move(in := 1, out1 => "DB251_ProgramDisplay".Display.RopeUnit7_1)
   END_RUNG
   RUNG wire#w1
      { S7_Templates := "SrcType := SInt" } LE_Contact(in1 := "DB251_ProgramDisplay".Display.RopeUnit7_1, in2 := 0)
   END_RUNG wire#w2
   RUNG wire#w1
      { S7_Templates := "SrcType := SInt" } GE_Contact(in1 := "DB251_ProgramDisplay".Display.RopeUnit8_1, in2 := 4)
      wire#w3
      { S7_GenerateENO := "TRUE" } Move(in := 1, out1 => "DB251_ProgramDisplay".Display.RopeUnit8_1)
   END_RUNG
   RUNG wire#w1
      { S7_Templates := "SrcType := SInt" } LE_Contact(in1 := "DB251_ProgramDisplay".Display.RopeUnit8_1, in2 := 0)
   END_RUNG wire#w3
   RUNG wire#w1
      { S7_Templates := "SrcType := SInt" } GE_Contact(in1 := "DB251_ProgramDisplay".Display.RopeUnit9_1, in2 := 4)
      wire#w4
      { S7_GenerateENO := "TRUE" } Move(in := 1, out1 => "DB251_ProgramDisplay".Display.RopeUnit9_1)
   END_RUNG
   RUNG wire#w1
      { S7_Templates := "SrcType := SInt" } LE_Contact(in1 := "DB251_ProgramDisplay".Display.RopeUnit9_1, in2 := 0)
   END_RUNG wire#w4
   RUNG wire#w1
      { S7_Templates := "SrcType := SInt" } GE_Contact(in1 := "DB251_ProgramDisplay".Display.RopeUnit10_1, in2 := 4)
      wire#w5
      { S7_GenerateENO := "TRUE" } Move(in := 1, out1 => "DB251_ProgramDisplay".Display.RopeUnit10_1)
   END_RUNG
   RUNG wire#w1
      { S7_Templates := "SrcType := SInt" } LE_Contact(in1 := "DB251_ProgramDisplay".Display.RopeUnit10_1, in2 := 0)
   END_RUNG wire#w5
   RUNG wire#w1
      { S7_Templates := "SrcType := SInt" } GE_Contact(in1 := "DB251_ProgramDisplay".Display.RopeUnit11_1, in2 := 4)
      wire#w6
      { S7_GenerateENO := "TRUE" } Move(in := 1, out1 => "DB251_ProgramDisplay".Display.RopeUnit11_1)
   END_RUNG
   RUNG wire#w1
      { S7_Templates := "SrcType := SInt" } LE_Contact(in1 := "DB251_ProgramDisplay".Display.RopeUnit11_1, in2 := 0)
   END_RUNG wire#w6
   RUNG wire#w1
      { S7_Templates := "SrcType := SInt" } GE_Contact(in1 := "DB251_ProgramDisplay".Display.RopeUnit12_1, in2 := 4)
      wire#w7
      { S7_GenerateENO := "TRUE" } Move(in := 1, out1 => "DB251_ProgramDisplay".Display.RopeUnit12_1)
   END_RUNG
   RUNG wire#w1
      { S7_Templates := "SrcType := SInt" } LE_Contact(in1 := "DB251_ProgramDisplay".Display.RopeUnit12_1, in2 := 0)
   END_RUNG wire#w7
   // the same network as SCL:
   IF "On" AND (("DB251_ProgramDisplay".Display.RopeUnit7_1 >= 4) OR ("DB251_ProgramDisplay".Display.RopeUnit7_1 <= 0)) THEN
       "DB251_ProgramDisplay".Display.RopeUnit7_1 := 1;
   END_IF;
   IF "On" AND (("DB251_ProgramDisplay".Display.RopeUnit8_1 >= 4) OR ("DB251_ProgramDisplay".Display.RopeUnit8_1 <= 0)) THEN
       "DB251_ProgramDisplay".Display.RopeUnit8_1 := 1;
   END_IF;
   IF "On" AND (("DB251_ProgramDisplay".Display.RopeUnit9_1 >= 4) OR ("DB251_ProgramDisplay".Display.RopeUnit9_1 <= 0)) THEN
       "DB251_ProgramDisplay".Display.RopeUnit9_1 := 1;
   END_IF;
   IF "On" AND (("DB251_ProgramDisplay".Display.RopeUnit10_1 >= 4) OR ("DB251_ProgramDisplay".Display.RopeUnit10_1 <= 0)) THEN
       "DB251_ProgramDisplay".Display.RopeUnit10_1 := 1;
   END_IF;
   IF "On" AND (("DB251_ProgramDisplay".Display.RopeUnit11_1 >= 4) OR ("DB251_ProgramDisplay".Display.RopeUnit11_1 <= 0)) THEN
       "DB251_ProgramDisplay".Display.RopeUnit11_1 := 1;
   END_IF;
   IF "On" AND (("DB251_ProgramDisplay".Display.RopeUnit12_1 >= 4) OR ("DB251_ProgramDisplay".Display.RopeUnit12_1 <= 0)) THEN
       "DB251_ProgramDisplay".Display.RopeUnit12_1 := 1;
   END_IF;
END_REGION

REGION Network 48: Rope unit out of range (1-6)
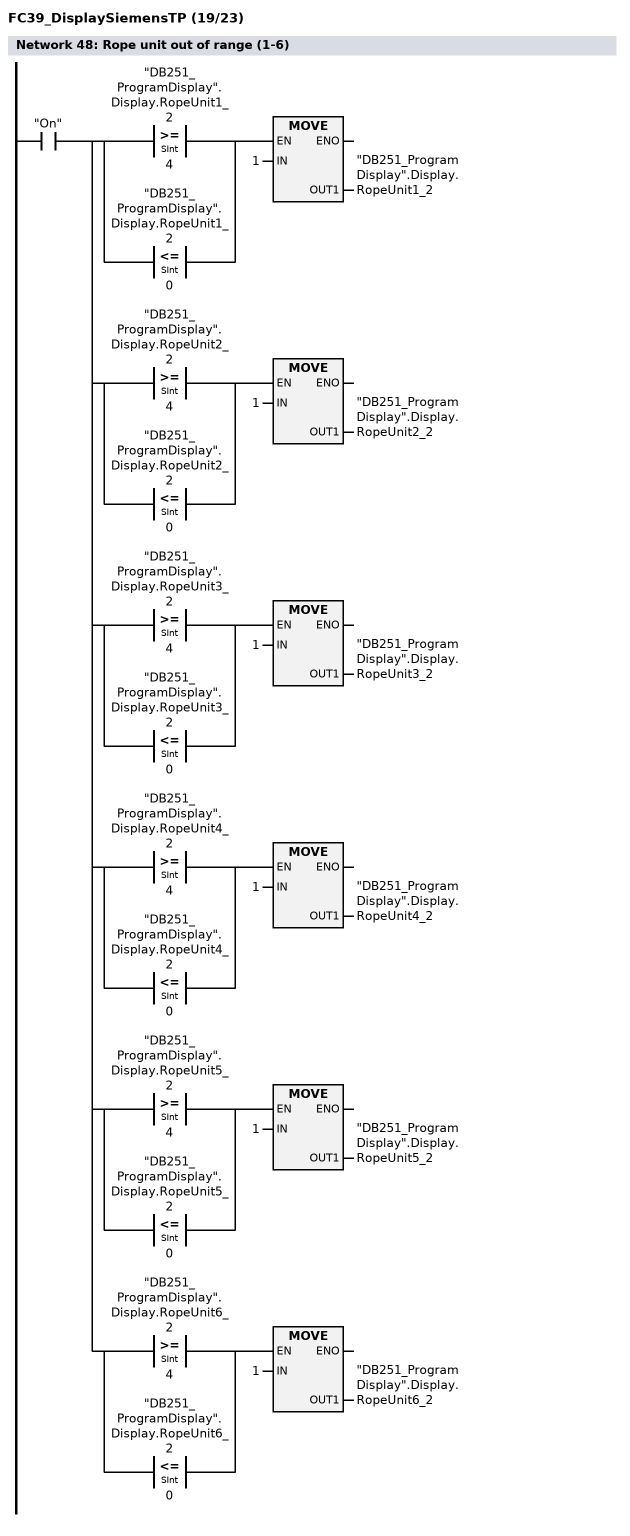
   RUNG wire#powerrail
      Contact( "On" )
      wire#w1
      { S7_Templates := "SrcType := SInt" } GE_Contact(in1 := "DB251_ProgramDisplay".Display.RopeUnit1_2, in2 := 4)
      wire#w2
      { S7_GenerateENO := "TRUE" } Move(in := 1, out1 => "DB251_ProgramDisplay".Display.RopeUnit1_2)
   END_RUNG
   RUNG wire#w1
      { S7_Templates := "SrcType := SInt" } LE_Contact(in1 := "DB251_ProgramDisplay".Display.RopeUnit1_2, in2 := 0)
   END_RUNG wire#w2
   RUNG wire#w1
      { S7_Templates := "SrcType := SInt" } GE_Contact(in1 := "DB251_ProgramDisplay".Display.RopeUnit2_2, in2 := 4)
      wire#w3
      { S7_GenerateENO := "TRUE" } Move(in := 1, out1 => "DB251_ProgramDisplay".Display.RopeUnit2_2)
   END_RUNG
   RUNG wire#w1
      { S7_Templates := "SrcType := SInt" } LE_Contact(in1 := "DB251_ProgramDisplay".Display.RopeUnit2_2, in2 := 0)
   END_RUNG wire#w3
   RUNG wire#w1
      { S7_Templates := "SrcType := SInt" } GE_Contact(in1 := "DB251_ProgramDisplay".Display.RopeUnit3_2, in2 := 4)
      wire#w4
      { S7_GenerateENO := "TRUE" } Move(in := 1, out1 => "DB251_ProgramDisplay".Display.RopeUnit3_2)
   END_RUNG
   RUNG wire#w1
      { S7_Templates := "SrcType := SInt" } LE_Contact(in1 := "DB251_ProgramDisplay".Display.RopeUnit3_2, in2 := 0)
   END_RUNG wire#w4
   RUNG wire#w1
      { S7_Templates := "SrcType := SInt" } GE_Contact(in1 := "DB251_ProgramDisplay".Display.RopeUnit4_2, in2 := 4)
      wire#w5
      { S7_GenerateENO := "TRUE" } Move(in := 1, out1 => "DB251_ProgramDisplay".Display.RopeUnit4_2)
   END_RUNG
   RUNG wire#w1
      { S7_Templates := "SrcType := SInt" } LE_Contact(in1 := "DB251_ProgramDisplay".Display.RopeUnit4_2, in2 := 0)
   END_RUNG wire#w5
   RUNG wire#w1
      { S7_Templates := "SrcType := SInt" } GE_Contact(in1 := "DB251_ProgramDisplay".Display.RopeUnit5_2, in2 := 4)
      wire#w6
      { S7_GenerateENO := "TRUE" } Move(in := 1, out1 => "DB251_ProgramDisplay".Display.RopeUnit5_2)
   END_RUNG
   RUNG wire#w1
      { S7_Templates := "SrcType := SInt" } LE_Contact(in1 := "DB251_ProgramDisplay".Display.RopeUnit5_2, in2 := 0)
   END_RUNG wire#w6
   RUNG wire#w1
      { S7_Templates := "SrcType := SInt" } GE_Contact(in1 := "DB251_ProgramDisplay".Display.RopeUnit6_2, in2 := 4)
      wire#w7
      { S7_GenerateENO := "TRUE" } Move(in := 1, out1 => "DB251_ProgramDisplay".Display.RopeUnit6_2)
   END_RUNG
   RUNG wire#w1
      { S7_Templates := "SrcType := SInt" } LE_Contact(in1 := "DB251_ProgramDisplay".Display.RopeUnit6_2, in2 := 0)
   END_RUNG wire#w7
   // the same network as SCL:
   IF "On" AND (("DB251_ProgramDisplay".Display.RopeUnit1_2 >= 4) OR ("DB251_ProgramDisplay".Display.RopeUnit1_2 <= 0)) THEN
       "DB251_ProgramDisplay".Display.RopeUnit1_2 := 1;
   END_IF;
   IF "On" AND (("DB251_ProgramDisplay".Display.RopeUnit2_2 >= 4) OR ("DB251_ProgramDisplay".Display.RopeUnit2_2 <= 0)) THEN
       "DB251_ProgramDisplay".Display.RopeUnit2_2 := 1;
   END_IF;
   IF "On" AND (("DB251_ProgramDisplay".Display.RopeUnit3_2 >= 4) OR ("DB251_ProgramDisplay".Display.RopeUnit3_2 <= 0)) THEN
       "DB251_ProgramDisplay".Display.RopeUnit3_2 := 1;
   END_IF;
   IF "On" AND (("DB251_ProgramDisplay".Display.RopeUnit4_2 >= 4) OR ("DB251_ProgramDisplay".Display.RopeUnit4_2 <= 0)) THEN
       "DB251_ProgramDisplay".Display.RopeUnit4_2 := 1;
   END_IF;
   IF "On" AND (("DB251_ProgramDisplay".Display.RopeUnit5_2 >= 4) OR ("DB251_ProgramDisplay".Display.RopeUnit5_2 <= 0)) THEN
       "DB251_ProgramDisplay".Display.RopeUnit5_2 := 1;
   END_IF;
   IF "On" AND (("DB251_ProgramDisplay".Display.RopeUnit6_2 >= 4) OR ("DB251_ProgramDisplay".Display.RopeUnit6_2 <= 0)) THEN
       "DB251_ProgramDisplay".Display.RopeUnit6_2 := 1;
   END_IF;
END_REGION

REGION Network 49: Rope unit out of range (7-12)
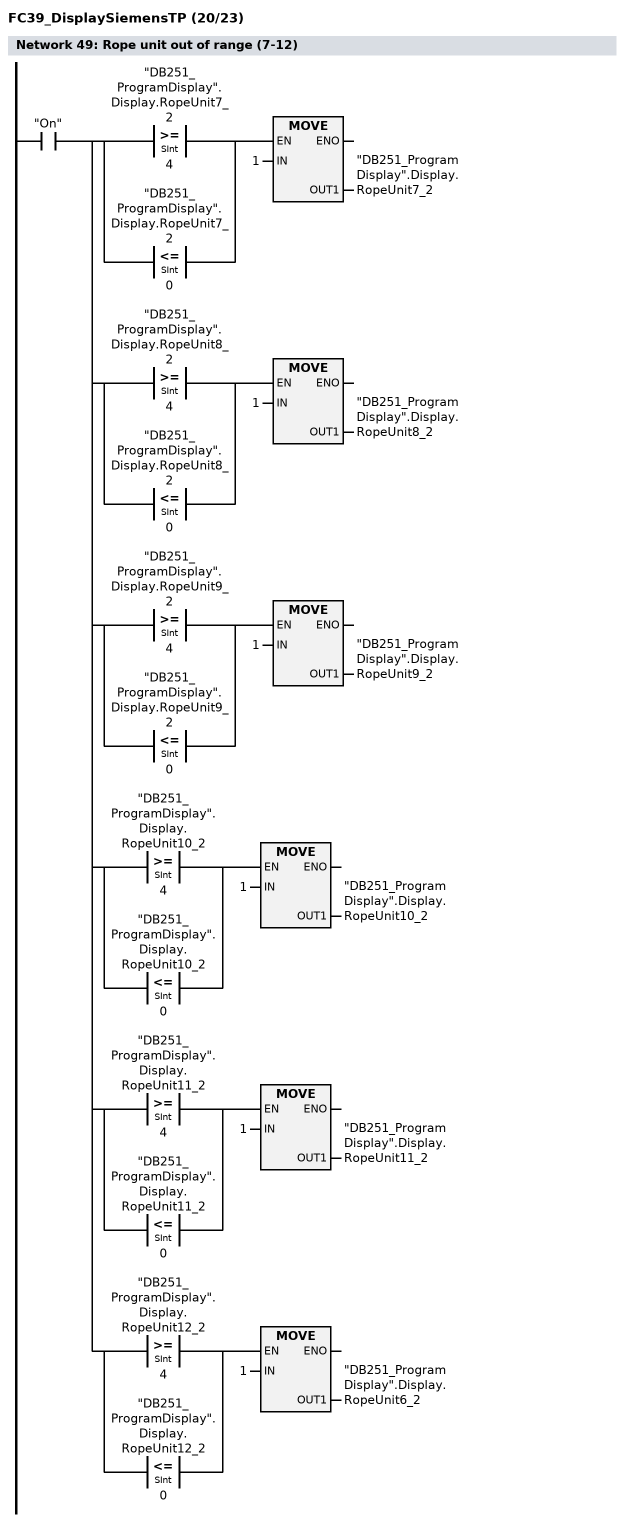
   RUNG wire#powerrail
      Contact( "On" )
      wire#w1
      { S7_Templates := "SrcType := SInt" } GE_Contact(in1 := "DB251_ProgramDisplay".Display.RopeUnit7_2, in2 := 4)
      wire#w2
      { S7_GenerateENO := "TRUE" } Move(in := 1, out1 => "DB251_ProgramDisplay".Display.RopeUnit7_2)
   END_RUNG
   RUNG wire#w1
      { S7_Templates := "SrcType := SInt" } LE_Contact(in1 := "DB251_ProgramDisplay".Display.RopeUnit7_2, in2 := 0)
   END_RUNG wire#w2
   RUNG wire#w1
      { S7_Templates := "SrcType := SInt" } GE_Contact(in1 := "DB251_ProgramDisplay".Display.RopeUnit8_2, in2 := 4)
      wire#w3
      { S7_GenerateENO := "TRUE" } Move(in := 1, out1 => "DB251_ProgramDisplay".Display.RopeUnit8_2)
   END_RUNG
   RUNG wire#w1
      { S7_Templates := "SrcType := SInt" } LE_Contact(in1 := "DB251_ProgramDisplay".Display.RopeUnit8_2, in2 := 0)
   END_RUNG wire#w3
   RUNG wire#w1
      { S7_Templates := "SrcType := SInt" } GE_Contact(in1 := "DB251_ProgramDisplay".Display.RopeUnit9_2, in2 := 4)
      wire#w4
      { S7_GenerateENO := "TRUE" } Move(in := 1, out1 => "DB251_ProgramDisplay".Display.RopeUnit9_2)
   END_RUNG
   RUNG wire#w1
      { S7_Templates := "SrcType := SInt" } LE_Contact(in1 := "DB251_ProgramDisplay".Display.RopeUnit9_2, in2 := 0)
   END_RUNG wire#w4
   RUNG wire#w1
      { S7_Templates := "SrcType := SInt" } GE_Contact(in1 := "DB251_ProgramDisplay".Display.RopeUnit10_2, in2 := 4)
      wire#w5
      { S7_GenerateENO := "TRUE" } Move(in := 1, out1 => "DB251_ProgramDisplay".Display.RopeUnit10_2)
   END_RUNG
   RUNG wire#w1
      { S7_Templates := "SrcType := SInt" } LE_Contact(in1 := "DB251_ProgramDisplay".Display.RopeUnit10_2, in2 := 0)
   END_RUNG wire#w5
   RUNG wire#w1
      { S7_Templates := "SrcType := SInt" } GE_Contact(in1 := "DB251_ProgramDisplay".Display.RopeUnit11_2, in2 := 4)
      wire#w6
      { S7_GenerateENO := "TRUE" } Move(in := 1, out1 => "DB251_ProgramDisplay".Display.RopeUnit11_2)
   END_RUNG
   RUNG wire#w1
      { S7_Templates := "SrcType := SInt" } LE_Contact(in1 := "DB251_ProgramDisplay".Display.RopeUnit11_2, in2 := 0)
   END_RUNG wire#w6
   RUNG wire#w1
      { S7_Templates := "SrcType := SInt" } GE_Contact(in1 := "DB251_ProgramDisplay".Display.RopeUnit12_2, in2 := 4)
      wire#w7
      { S7_GenerateENO := "TRUE" } Move(in := 1, out1 => "DB251_ProgramDisplay".Display.RopeUnit6_2)
   END_RUNG
   RUNG wire#w1
      { S7_Templates := "SrcType := SInt" } LE_Contact(in1 := "DB251_ProgramDisplay".Display.RopeUnit12_2, in2 := 0)
   END_RUNG wire#w7
   // the same network as SCL:
   IF "On" AND (("DB251_ProgramDisplay".Display.RopeUnit7_2 >= 4) OR ("DB251_ProgramDisplay".Display.RopeUnit7_2 <= 0)) THEN
       "DB251_ProgramDisplay".Display.RopeUnit7_2 := 1;
   END_IF;
   IF "On" AND (("DB251_ProgramDisplay".Display.RopeUnit8_2 >= 4) OR ("DB251_ProgramDisplay".Display.RopeUnit8_2 <= 0)) THEN
       "DB251_ProgramDisplay".Display.RopeUnit8_2 := 1;
   END_IF;
   IF "On" AND (("DB251_ProgramDisplay".Display.RopeUnit9_2 >= 4) OR ("DB251_ProgramDisplay".Display.RopeUnit9_2 <= 0)) THEN
       "DB251_ProgramDisplay".Display.RopeUnit9_2 := 1;
   END_IF;
   IF "On" AND (("DB251_ProgramDisplay".Display.RopeUnit10_2 >= 4) OR ("DB251_ProgramDisplay".Display.RopeUnit10_2 <= 0)) THEN
       "DB251_ProgramDisplay".Display.RopeUnit10_2 := 1;
   END_IF;
   IF "On" AND (("DB251_ProgramDisplay".Display.RopeUnit11_2 >= 4) OR ("DB251_ProgramDisplay".Display.RopeUnit11_2 <= 0)) THEN
       "DB251_ProgramDisplay".Display.RopeUnit11_2 := 1;
   END_IF;
   IF "On" AND (("DB251_ProgramDisplay".Display.RopeUnit12_2 >= 4) OR ("DB251_ProgramDisplay".Display.RopeUnit12_2 <= 0)) THEN
       "DB251_ProgramDisplay".Display.RopeUnit6_2 := 1;
   END_IF;
END_REGION

REGION Network 50: Define landmark to bottom for the last step
